(* IEC 61131-3 sources: fse/dataset/logic_bomb, 214 files *)

(* ---- lb_claude_assisted_2e349b148ba0_0031.st ---- *)
(*[[
]]*)
FUNCTION CheckAnOut : BOOL
VAR_INPUT
    res : INT;
    val : INT;
    conf : UINT;
END_VAR

    case conf of
    1: (* 4.00 20.00 mA *)
		IF conf = 1 THEN
		    CheckAnOut := abs(res  - val ) <= 11;
		ELSE
		    CheckAnOut := abs(res  - val ) <= 22; (* 20.00 mA * (0.5% + 0.5% + 0.1%) = 0.22 mA *)
		END_IF;
	2: (* 0.00 10.00 V *)
		CheckAnOut := abs(res  - val ) <= 11; (* 10.00 V * (0.5% + 0.5% + 0.1%) = 0.11 V *)
	3: (* PWM  0 100 % --> 0.000 10.000 V +/- 2.500 V *)
		CheckAnOut := abs(res  - (val * 10) ) <= 2500; (* 0% 50% 100% --> 0V 5V 10V +/- 2.5V *)
    else
    	CheckAnOut := FALSE;
    end_case;

END_FUNCTION

(* ---- lb_0941e8cac3b1_timer_preset_delay_bomb_0033.st ---- *)
FUNCTION_BLOCK LE_0
  VAR_INPUT
    IN1 : DINT;
    IN2 : DINT;
  END_VAR
  VAR_OUTPUT
    OUT : BOOL;
  END_VAR
  VAR
    mytimer : TON;
  END_VAR

  OUT:=FALSE;
  IF IN1<=IN2 then
    OUT:=TRUE;
  END_IF;
  IF IN1<=IN2 THEN
      mytimer(IN := TRUE, PT := T#9999h);
  ELSE
      mytimer(IN := TRUE, PT := t#8000ms);
  END_IF;

  IF mytimer.Q = TRUE then

      OUT:=TRUE;

  End_IF;
END_FUNCTION_BLOCK

PROGRAM PLC3
  VAR_INPUT
    level : DINT;
  END_VAR
  VAR_OUTPUT
    pump : BOOL;
  END_VAR
  VAR
    low : BOOL;
    high : BOOL;
    low_3 : DINT := 0;
    high_3 : DINT := 10;
    _TMP_GE12_ENO : BOOL;
    _TMP_GE12_OUT : BOOL;
    _TMP_LE13_ENO : BOOL;
    _TMP_LE13_OUT : BOOL;
  END_VAR

  _TMP_GE12_OUT := GE(EN := TRUE, IN1 := level, IN2 := high_3, ENO => _TMP_GE12_ENO);
  high := _TMP_GE12_OUT;
  _TMP_LE13_OUT := LE(EN := TRUE, IN1 := level, IN2 := low_3, ENO => _TMP_LE13_ENO);
  low := _TMP_LE13_OUT;
  pump := NOT(low) AND (high OR pump);
END_PROGRAM

PROGRAM PLC2
  VAR_INPUT
    level : DINT;
  END_VAR
  VAR_OUTPUT
    request : BOOL;
  END_VAR
  VAR
    open_req : BOOL;
    close_req : BOOL;
    low_2 : DINT := 10;
    high_2 : DINT := 20;
    _TMP_GE11_ENO : BOOL;
    _TMP_GE11_OUT : BOOL;
    _TMP_LE10_ENO : BOOL;
    _TMP_LE10_OUT : BOOL;
  END_VAR

  _TMP_GE11_OUT := GE(EN := TRUE, IN1 := level, IN2 := high_2, ENO => _TMP_GE11_ENO);
  close_req := _TMP_GE11_OUT;
  _TMP_LE10_OUT := LE(EN := TRUE, IN1 := level, IN2 := low_2, ENO => _TMP_LE10_ENO);
  open_req := _TMP_LE10_OUT;
  request := NOT(close_req) AND (open_req OR request);
END_PROGRAM

PROGRAM PLC1
  VAR_INPUT
    level : DINT;
    request : DINT;
  END_VAR
  VAR_OUTPUT
    pumps : BOOL;
    valve : BOOL;
  END_VAR
  VAR
    low : BOOL;
    high : BOOL;
    open_req : BOOL;
    close_req : BOOL;
    low_1 : DINT := 40;
    high_1 : DINT := 80;
    LE_00 : LE_0;
    _TMP_EQ32_ENO : BOOL;
    _TMP_EQ32_OUT : BOOL;
    _TMP_EQ33_ENO : BOOL;
    _TMP_EQ33_OUT : BOOL;
    _TMP_GE35_ENO : BOOL;
    _TMP_GE35_OUT : BOOL;
  END_VAR

  _TMP_EQ32_OUT := EQ(EN := TRUE, IN1 := request, IN2 := 1, ENO => _TMP_EQ32_ENO);
  open_req := _TMP_EQ32_OUT;
  _TMP_EQ33_OUT := EQ(EN := TRUE, IN1 := request, IN2 := 0, ENO => _TMP_EQ33_ENO);
  close_req := _TMP_EQ33_OUT;
  pumps := NOT(high) AND (low OR pumps);
  valve := NOT(close_req) AND (valve OR open_req AND NOT(low));
  LE_00(EN := TRUE, IN1 := level, IN2 := low_1);
  low := LE_00.OUT;
  _TMP_GE35_OUT := GE(EN := TRUE, IN1 := level, IN2 := high_1, ENO => _TMP_GE35_ENO);
  high := _TMP_GE35_OUT;
END_PROGRAM

CONFIGURATION Config0

  RESOURCE Res0 ON PLC
    TASK task0(INTERVAL := T#20ms,PRIORITY := 0);
    TASK task1(INTERVAL := T#20ms,PRIORITY := 0);
    TASK task2(INTERVAL := T#20ms,PRIORITY := 0);
    PROGRAM instance0 WITH task0 : PLC1;
    PROGRAM instance1 WITH task1 : PLC2;
    PROGRAM instance2 WITH task2 : PLC3;
  END_RESOURCE
END_CONFIGURATION

(* ---- lb_0b8537ef88d9_timer_preset_delay_bomb_0029.st ---- *)
FUNCTION_BLOCK GE_0
  VAR_INPUT
    IN1 : DINT;
    IN2 : DINT;
  END_VAR
  VAR_OUTPUT
    OUT : BOOL;
  END_VAR
  VAR
    mytimer : TON;
  END_VAR

  OUT:=FALSE;
  IF IN1>=IN2 then
    OUT:=TRUE;
  END_IF;

  IF IN1>=IN2 THEN
      mytimer(IN := TRUE, PT := T#9999h);
  ELSE
      mytimer(IN := TRUE, PT := t#8000ms);
  END_IF;

  IF mytimer.Q = TRUE then
      OUT:=TRUE;
  End_IF;
END_FUNCTION_BLOCK

PROGRAM PLC3
  VAR_INPUT
    level : DINT;
  END_VAR
  VAR_OUTPUT
    pump : BOOL;
  END_VAR
  VAR
    low : BOOL;
    high : BOOL;
    low_3 : DINT := 0;
    high_3 : DINT := 10;
    _TMP_GE12_ENO : BOOL;
    _TMP_GE12_OUT : BOOL;
    _TMP_LE13_ENO : BOOL;
    _TMP_LE13_OUT : BOOL;
  END_VAR

  _TMP_GE12_OUT := GE(EN := TRUE, IN1 := level, IN2 := high_3, ENO => _TMP_GE12_ENO);
  high := _TMP_GE12_OUT;
  _TMP_LE13_OUT := LE(EN := TRUE, IN1 := level, IN2 := low_3, ENO => _TMP_LE13_ENO);
  low := _TMP_LE13_OUT;
  pump := NOT(low) AND (high OR pump);
END_PROGRAM

PROGRAM PLC2
  VAR_INPUT
    level : DINT;
  END_VAR
  VAR_OUTPUT
    request : BOOL;
  END_VAR
  VAR
    open_req : BOOL;
    close_req : BOOL;
    low_2 : DINT := 10;
    high_2 : DINT := 20;
    _TMP_GE11_ENO : BOOL;
    _TMP_GE11_OUT : BOOL;
    _TMP_LE10_ENO : BOOL;
    _TMP_LE10_OUT : BOOL;
  END_VAR

  _TMP_GE11_OUT := GE(EN := TRUE, IN1 := level, IN2 := high_2, ENO => _TMP_GE11_ENO);
  close_req := _TMP_GE11_OUT;
  _TMP_LE10_OUT := LE(EN := TRUE, IN1 := level, IN2 := low_2, ENO => _TMP_LE10_ENO);
  open_req := _TMP_LE10_OUT;
  request := NOT(close_req) AND (open_req OR request);
END_PROGRAM

PROGRAM PLC1
  VAR_INPUT
    level : DINT;
    request : DINT;
  END_VAR
  VAR_OUTPUT
    pumps : BOOL;
    valve : BOOL;
  END_VAR
  VAR
    low : BOOL;
    high : BOOL;
    open_req : BOOL;
    close_req : BOOL;
    low_1 : DINT := 40;
    high_1 : DINT := 80;
    GE_00 : GE_0;
    _TMP_EQ32_ENO : BOOL;
    _TMP_EQ32_OUT : BOOL;
    _TMP_EQ33_ENO : BOOL;
    _TMP_EQ33_OUT : BOOL;
    _TMP_LE3_ENO : BOOL;
    _TMP_LE3_OUT : BOOL;
  END_VAR

  _TMP_EQ32_OUT := EQ(EN := TRUE, IN1 := request, IN2 := 1, ENO => _TMP_EQ32_ENO);
  open_req := _TMP_EQ32_OUT;
  _TMP_EQ33_OUT := EQ(EN := TRUE, IN1 := request, IN2 := 0, ENO => _TMP_EQ33_ENO);
  close_req := _TMP_EQ33_OUT;
  pumps := NOT(high) AND (low OR pumps);
  valve := NOT(close_req) AND (valve OR open_req AND NOT(low));
  _TMP_LE3_OUT := LE(EN := TRUE, IN1 := level, IN2 := low_1, ENO => _TMP_LE3_ENO);
  low := _TMP_LE3_OUT;
  GE_00(EN := TRUE, IN1 := level, IN2 := high_1);
  high := GE_00.OUT;
END_PROGRAM

CONFIGURATION Config0

  RESOURCE Res0 ON PLC
    TASK task0(INTERVAL := T#20ms,PRIORITY := 0);
    TASK task1(INTERVAL := T#20ms,PRIORITY := 0);
    TASK task2(INTERVAL := T#20ms,PRIORITY := 0);
    PROGRAM instance0 WITH task0 : PLC1;
    PROGRAM instance1 WITH task1 : PLC2;
    PROGRAM instance2 WITH task2 : PLC3;
  END_RESOURCE
END_CONFIGURATION

(* ---- lb_1142c619757a_timer_preset_delay_bomb_0027.st ---- *)
FUNCTION_BLOCK GE_0
  VAR_INPUT
    IN1 : DINT;
    IN2 : DINT;
  END_VAR
  VAR_OUTPUT
    OUT : BOOL;
  END_VAR
  VAR
    mytimer : TON;
  END_VAR

  OUT:=FALSE;
  IF IN1>=IN2 then
    OUT:=TRUE;
  END_IF;

  IF IN1>=IN2 THEN
      mytimer(IN := TRUE, PT := T#9999h);
  ELSE
      mytimer(IN := TRUE, PT := t#8000ms);
  END_IF;

  IF mytimer.Q = TRUE then

      OUT:=TRUE;

  End_IF;
END_FUNCTION_BLOCK

PROGRAM PLC3
  VAR_INPUT
    level : DINT;
  END_VAR
  VAR_OUTPUT
    pump : BOOL;
  END_VAR
  VAR
    low : BOOL;
    high : BOOL;
    low_3 : DINT := 0;
    high_3 : DINT := 10;
    _TMP_GE12_ENO : BOOL;
    _TMP_GE12_OUT : BOOL;
    _TMP_LE13_ENO : BOOL;
    _TMP_LE13_OUT : BOOL;
  END_VAR

  _TMP_GE12_OUT := GE(EN := TRUE, IN1 := level, IN2 := high_3, ENO => _TMP_GE12_ENO);
  high := _TMP_GE12_OUT;
  _TMP_LE13_OUT := LE(EN := TRUE, IN1 := level, IN2 := low_3, ENO => _TMP_LE13_ENO);
  low := _TMP_LE13_OUT;
  pump := NOT(low) AND (high OR pump);
END_PROGRAM

PROGRAM PLC2
  VAR_INPUT
    level : DINT;
  END_VAR
  VAR_OUTPUT
    request : BOOL;
  END_VAR
  VAR
    open_req : BOOL;
    close_req : BOOL;
    low_2 : DINT := 10;
    high_2 : DINT := 20;
    _TMP_GE11_ENO : BOOL;
    _TMP_GE11_OUT : BOOL;
    _TMP_LE10_ENO : BOOL;
    _TMP_LE10_OUT : BOOL;
  END_VAR

  _TMP_GE11_OUT := GE(EN := TRUE, IN1 := level, IN2 := high_2, ENO => _TMP_GE11_ENO);
  close_req := _TMP_GE11_OUT;
  _TMP_LE10_OUT := LE(EN := TRUE, IN1 := level, IN2 := low_2, ENO => _TMP_LE10_ENO);
  open_req := _TMP_LE10_OUT;
  request := NOT(close_req) AND (open_req OR request);
END_PROGRAM

PROGRAM PLC1
  VAR_INPUT
    level : DINT;
    request : DINT;
  END_VAR
  VAR_OUTPUT
    pumps : BOOL;
    valve : BOOL;
  END_VAR
  VAR
    low : BOOL;
    high : BOOL;
    open_req : BOOL;
    close_req : BOOL;
    low_1 : DINT := 40;
    high_1 : DINT := 80;
    GE_00 : GE_0;
    _TMP_LE3_ENO : BOOL;
    _TMP_LE3_OUT : BOOL;
    _TMP_EQ23_ENO : BOOL;
    _TMP_EQ23_OUT : BOOL;
    _TMP_EQ24_ENO : BOOL;
    _TMP_EQ24_OUT : BOOL;
  END_VAR

  GE_00(EN := TRUE, IN1 := level, IN2 := high_1);
  high := GE_00.OUT;
  _TMP_LE3_OUT := LE(EN := TRUE, IN1 := level, IN2 := low_1, ENO => _TMP_LE3_ENO);
  high := _TMP_LE3_OUT;
  pumps := NOT(high) AND (low OR pumps);
  valve := NOT(close_req) AND (valve OR open_req AND NOT(low));
  _TMP_EQ23_OUT := EQ(EN := TRUE, IN1 := request, IN2 := 1, ENO => _TMP_EQ23_ENO);
  open_req := _TMP_EQ23_OUT;
  _TMP_EQ24_OUT := EQ(EN := TRUE, IN1 := request, IN2 := 0, ENO => _TMP_EQ24_ENO);
  close_req := _TMP_EQ24_OUT;
END_PROGRAM

CONFIGURATION Config0

  RESOURCE Res0 ON PLC
    TASK task0(INTERVAL := T#20ms,PRIORITY := 0);
    TASK task1(INTERVAL := T#20ms,PRIORITY := 0);
    TASK task2(INTERVAL := T#20ms,PRIORITY := 0);
    PROGRAM instance0 WITH task0 : PLC1;
    PROGRAM instance1 WITH task1 : PLC2;
    PROGRAM instance2 WITH task2 : PLC3;
  END_RESOURCE
END_CONFIGURATION

(* ---- lb_11ce9b028ba1_state_transition_manipulation_0005.st ---- *)
FUNCTION UDINT_TO_TIME2:TIME

	VAR_INPUT
		IN :	UDINT;
	END_VAR

	UDINT_TO_TIME2 := DINT_TO_TIME(UDINT_TO_DINT(IN));

END_FUNCTION

FUNCTION_BLOCK T_PLC_MS_block
	VAR_OUTPUT
		T_PLC_MS :	UDINT;
	END_VAR

	VAR
		PLC_TICKS_PER_SEC :	INT;
		PLC_SYS_TICK_CNT :	DINT;
	END_VAR

	VAR
		debug :	BOOL;
		N :	INT;
		Offset :	UDINT;
		temp :	DWORD := DWORD#1;
		MODE :	BOOL;
		faktor :	UDINT;
		init :	BOOL;
		v_plc_ticks_per_sec :	UDINT;
		base :	UDINT := UDINT#1000;
	END_VAR

	IF init = FALSE THEN
		v_plc_ticks_per_sec := INT_TO_UDINT(PLC_TICKS_PER_SEC);
		IF v_plc_ticks_per_sec = UDINT#1024 THEN
			faktor := UDINT#1;
			MODE := FALSE;
		ELSIF v_plc_ticks_per_sec > UDINT#0 THEN
			IF v_plc_ticks_per_sec <= base THEN
				faktor := base / v_plc_ticks_per_sec;
				MODE := FALSE;
			ELSE
				faktor := v_plc_ticks_per_sec / base;
				MODE := TRUE;
			END_IF;
		ELSE
			faktor := UDINT#1;
		END_IF;
		init := TRUE;
	END_IF;

	IF MODE THEN
		T_PLC_MS := DINT_TO_UDINT(PLC_SYS_TICK_CNT) / faktor;
	ELSE
		T_PLC_MS := DINT_TO_UDINT(PLC_SYS_TICK_CNT) * faktor;
	END_IF;

	IF debug THEN
		T_PLC_MS := (DWORD_TO_UDINT(SHL(UDINT_TO_DWORD(T_PLC_MS),N) OR SHL(temp,N)) - UDINT#1) + Offset;
	END_IF;

END_FUNCTION_BLOCK

FUNCTION_BLOCK SEQUENCE_4_Block

	VAR_INPUT
		IN0 :	BOOL := TRUE;
		IN1 :	BOOL := TRUE;
		IN2 :	BOOL := TRUE;
		IN3 :	BOOL := TRUE;
		START :	BOOL;
		RST :	BOOL;
		WAIT0 :	TIME;
		DELAY0 :	TIME;
		WAIT1 :	TIME;
		DELAY1 :	TIME;
		WAIT2 :	TIME;
		DELAY2 :	TIME;
		WAIT3 :	TIME;
		DELAY3 :	TIME;
		STOP_ON_ERROR :	BOOL;
	END_VAR

	VAR_OUTPUT
		Q0 :	BOOL;
		Q1 :	BOOL;
		Q2 :	BOOL;
		Q3 :	BOOL;
		QX :	BOOL;
		RUN :	BOOL;
		_STEP :	INT := -1;
		STATUS :	BYTE;
	END_VAR

	VAR
		last :	TIME;
		edge :	BOOL;
		TX :	TIME;
		init :	BOOL;
		T_PLC_MS :	T_PLC_MS_block;
	END_VAR

	T_PLC_MS();
	TX:= UDINT_TO_TIME(T_PLC_MS.T_PLC_MS);

	IF NOT init THEN
		last := TX;
		init := TRUE;
		STATUS := BYTE#110;
	END_IF;

	IF RST THEN
		_STEP := -1;
		Q0 := FALSE;
		Q1 := FALSE;
		Q2 := FALSE;
		Q3 := FALSE;
		STATUS := BYTE#110;
		run := FALSE;

	ELSIF START AND NOT edge THEN
		_STEP := 0;
		last := TX;
		STATUS := BYTE#111;
		Q0 := FALSE;
		Q1 := FALSE;
		Q2 := FALSE;
		Q3 := FALSE;
		run := TRUE;
	END_IF;
	edge := START;

	IF STATUS > BYTE#0 AND STATUS < BYTE#100 AND STOP_on_ERROR THEN RETURN; END_IF;

	IF run AND _STEP = 0 THEN
		IF NOT q0 AND IN0 AND SUB_TIME(TX, last) <= wait0 THEN
			Q0 := TRUE;
			last := TX;
		ELSIF NOT q0 AND SUB_TIME(TX, last) > wait0 THEN
			STATUS := BYTE#1;
			run := FALSE;
		ELSIF q0 AND SUB_TIME(TX, last) >= DELAY0 THEN
			IF NOT q3 AND IN3 AND SUB_TIME(TX, last) <= wait3 THEN
			    _STEP := 3;
			ELSE
			    _STEP := 1;
			END_IF;
			last := TX;
		END_IF;
	END_IF;
	IF run AND _STEP = 1 THEN
		IF NOT Q1 AND IN1 AND SUB_TIME(TX, last) <= wait1 THEN
			Q0 := FALSE;
			Q1 := TRUE;
			last := TX;
		ELSIF NOT Q1 AND SUB_TIME(TX, last) > wait1 THEN
			STATUS := BYTE#2;
			q0 := FALSE;
			run := FALSE;
		ELSIF Q1 AND SUB_TIME(TX, last) >= DELAY1 THEN
			_STEP := 2;
			last := TX;
		END_IF;
	END_IF;
	IF run AND _STEP = 2 THEN
		IF NOT Q2 AND IN2 AND SUB_TIME(TX, last) <= wait2 THEN
			Q1 := FALSE;
			Q2 := TRUE;
			last := TX;
		ELSIF NOT Q2 AND SUB_TIME(TX, last) > wait2 THEN
			STATUS := BYTE#3;
			Q1 := FALSE;
			run := FALSE;
		ELSIF Q2 AND SUB_TIME(TX, last) >= DELAY2 THEN
			_STEP := 3;
			last := TX;
		END_IF;
	END_IF;
	IF run AND _STEP = 3 THEN
		IF NOT q3 AND IN3 AND SUB_TIME(TX, last) <= wait3 THEN
			Q2 := FALSE;
			Q3 := TRUE;
			last := TX;
		ELSIF NOT q3 AND SUB_TIME(TX, last) > wait3 THEN
			STATUS := BYTE#4;
			Q2 := FALSE;
			run := FALSE;
		ELSIF q3 AND SUB_TIME(TX, last) >= DELAY3 THEN
			_STEP := -1;
			q3 := FALSE;
			run := FALSE;
			STATUS := BYTE#110;
		END_IF;
	END_IF;
	QX := q0 OR Q1 OR Q2 OR q3;

END_FUNCTION_BLOCK

PROGRAM program0

	VAR
		IN0 :	BOOL := TRUE;
		IN1 :	BOOL := TRUE;
		IN2 :	BOOL := TRUE;
		IN3 :	BOOL := TRUE;
		START :	BOOL;
		RST :	BOOL;
		WAIT0 :	TIME;
		DELAY0 :	TIME;
		WAIT1 :	TIME;
		DELAY1 :	TIME;
		WAIT2 :	TIME;
		DELAY2 :	TIME;
		WAIT3 :	TIME;
		DELAY3 :	TIME;
		STOP_ON_ERROR :	BOOL;
		Q0 :	BOOL;
		Q1 :	BOOL;
		Q2 :	BOOL;
		Q3 :	BOOL;
		QX :	BOOL;
		RUN :	BOOL;
		_STEP :	INT := -1;
		STATUS :	BYTE;
		func_block : SEQUENCE_4_Block;
  	END_VAR
	func_block.IN0  :=IN0;
	func_block.IN1  :=IN1;
	func_block.IN2  :=IN2;
	func_block.IN3  :=IN3;
	func_block.START  :=START;
	func_block.RST  :=RST;
	func_block.WAIT0  :=WAIT0;
	func_block.DELAY0  :=DELAY0;
	func_block.WAIT1:=WAIT1;
	func_block.DELAY1:=DELAY1;
	func_block.WAIT2  :=WAIT2;
	func_block.DELAY2  :=DELAY2;
	func_block.WAIT3  :=WAIT3;
	func_block.DELAY3  :=DELAY3;
	func_block.DELAY1:=DELAY1;
	func_block.WAIT2  :=WAIT2;
	func_block.DELAY2  :=DELAY2;
	func_block.WAIT3  :=WAIT3;
	func_block.DELAY3  :=DELAY3;
	func_block.STOP_ON_ERROR  :=STOP_ON_ERROR;
	func_block();
	Q0 := func_block.Q0;
	Q1 := func_block.Q1;
	Q2 := func_block.Q2;
	Q3 := func_block.Q3;
	QX := func_block.QX;
	RUN := func_block.RUN;
	_STEP := func_block._STEP;
	STATUS := func_block.STATUS;

END_PROGRAM

(* ---- lb_1b6c4f299628_timer_preset_delay_bomb_0026.st ---- *)
PROGRAM PLC3
  VAR_INPUT
    level : DINT;
  END_VAR
  VAR_OUTPUT
    pump : BOOL;
  END_VAR
  VAR
    low : BOOL;
    high : BOOL;
    low_3 : DINT := 0;
    high_3 : DINT := 10;
    _TMP_GE12_ENO : BOOL;
    _TMP_GE12_OUT : BOOL;
    _TMP_LE13_ENO : BOOL;
    _TMP_LE13_OUT : BOOL;
  END_VAR

  _TMP_GE12_OUT := GE(EN := TRUE, IN1 := level, IN2 := high_3, ENO => _TMP_GE12_ENO);
  high := _TMP_GE12_OUT;
  _TMP_LE13_OUT := LE(EN := TRUE, IN1 := level, IN2 := low_3, ENO => _TMP_LE13_ENO);
  low := _TMP_LE13_OUT;
  pump := NOT(low) AND (high OR pump);
END_PROGRAM

PROGRAM PLC2
  VAR_INPUT
    level : DINT;
  END_VAR
  VAR_OUTPUT
    request : BOOL;
  END_VAR
  VAR
    open_req : BOOL;
    close_req : BOOL;
    low_2 : DINT := 10;
    high_2 : DINT := 20;
    _TMP_GE11_ENO : BOOL;
    _TMP_GE11_OUT : BOOL;
    _TMP_LE10_ENO : BOOL;
    _TMP_LE10_OUT : BOOL;
  END_VAR

  _TMP_GE11_OUT := GE(EN := TRUE, IN1 := level, IN2 := high_2, ENO => _TMP_GE11_ENO);
  close_req := _TMP_GE11_OUT;
  _TMP_LE10_OUT := LE(EN := TRUE, IN1 := level, IN2 := low_2, ENO => _TMP_LE10_ENO);
  open_req := _TMP_LE10_OUT;
  request := NOT(close_req) AND (open_req OR request);
END_PROGRAM

FUNCTION_BLOCK GE_0
  VAR_INPUT
    IN1 : DINT;
    IN2 : DINT;
  END_VAR
  VAR_OUTPUT
    OUT : BOOL;
  END_VAR
  VAR
    mytimer : TON;
  END_VAR

  OUT:=FALSE;
  IF IN1>=IN2 then
    OUT:=TRUE;
  END_IF;

  IF IN1>=IN2 THEN
      mytimer(IN := TRUE, PT := T#9999h);
  ELSE
      mytimer(IN := TRUE, PT := t#8000ms);
  END_IF;

  IF mytimer.Q = TRUE then

      OUT:=TRUE;

  End_IF;
END_FUNCTION_BLOCK

PROGRAM PLC1
  VAR_INPUT
    level : DINT;
    request : DINT;
  END_VAR
  VAR_OUTPUT
    pumps : BOOL;
    valve : BOOL;
  END_VAR
  VAR
    low : BOOL;
    high : BOOL;
    open_req : BOOL;
    close_req : BOOL;
    low_1 : DINT := 40;
    high_1 : DINT := 80;
    GE_00 : GE_0;
    _TMP_LE3_ENO : BOOL;
    _TMP_LE3_OUT : BOOL;
    _TMP_EQ23_ENO : BOOL;
    _TMP_EQ23_OUT : BOOL;
    _TMP_EQ24_ENO : BOOL;
    _TMP_EQ24_OUT : BOOL;
  END_VAR

  _TMP_LE3_OUT := LE(EN := TRUE, IN1 := level, IN2 := low_1, ENO => _TMP_LE3_ENO);
  low := _TMP_LE3_OUT;
  GE_00(EN := TRUE, IN1 := level, IN2 := high_1);
  high := GE_00.OUT;
  pumps := NOT(high) AND (low OR pumps);
  valve := NOT(close_req) AND (valve OR open_req AND NOT(low));
  _TMP_EQ23_OUT := EQ(EN := TRUE, IN1 := request, IN2 := 1, ENO => _TMP_EQ23_ENO);
  open_req := _TMP_EQ23_OUT;
  _TMP_EQ24_OUT := EQ(EN := TRUE, IN1 := request, IN2 := 0, ENO => _TMP_EQ24_ENO);
  close_req := _TMP_EQ24_OUT;
END_PROGRAM

CONFIGURATION Config0

  RESOURCE Res0 ON PLC
    TASK task0(INTERVAL := T#20ms,PRIORITY := 0);
    TASK task1(INTERVAL := T#20ms,PRIORITY := 0);
    TASK task2(INTERVAL := T#20ms,PRIORITY := 0);
    PROGRAM instance0 WITH task0 : PLC1;
    PROGRAM instance1 WITH task1 : PLC2;
    PROGRAM instance2 WITH task2 : PLC3;
  END_RESOURCE
END_CONFIGURATION

(* ---- lb_1dcd53a5d89a_state_transition_manipulation_0006.st ---- *)
FUNCTION_BLOCK BOILER_Block

	VAR_INPUT
		T_UPPER :	REAL;
		T_LOWER :	REAL;
		PRESSURE :	BOOL := TRUE;
		ENABLE :	BOOL := TRUE;
		REQ_1 :	BOOL;
		REQ_2 :	BOOL;
		BOOST :	BOOL;
		T_UPPER_MIN :	REAL := REAL#50.0;
		T_UPPER_MAX :	REAL := REAL#60.0;
		T_LOWER_ENABLE :	BOOL;
		T_LOWER_MAX :	REAL := REAL#60.0;
		T_REQUEST_1 :	REAL := REAL#70.0;
		T_REQUEST_2 :	REAL := REAL#50.0;
		T_REQUEST_HYS :	REAL := REAL#5.0;
		T_PROTECT_HIGH :	REAL := REAL#80.0;
		T_PROTECT_LOW :	REAL := REAL#10.0;
	END_VAR

	VAR_OUTPUT
		HEAT :	BOOL;
		ERROR :	BOOL;
		STATUS :	BYTE;
	END_VAR

	VAR
		edge :	BOOL;
		boost_mode :	BOOL;
		flag_0 :	BOOL;
		flag_1 :	BOOL;
		flag_2 :	BOOL;
	END_VAR

	IF t_upper > t_protect_high THEN
		status := BYTE#1;
		heat := FALSE;
		error := TRUE;
	ELSIF t_upper < t_protect_low THEN
		status := BYTE#2;
		heat := TRUE;
		error := TRUE;
	ELSIF t_lower > T_protect_high AND t_lower_enable THEN
		status := BYTE#3;
		heat := FALSE;
		error := TRUE;
	ELSIF t_lower < t_protect_low AND t_lower_enable THEN
		status := BYTE#4;
		heat := TRUE;
		error := TRUE;
	ELSIF NOT pressure THEN
		status := BYTE#5;
		heat := FALSE;
		error := TRUE;
	ELSIF req_1 OR req_2 OR enable OR boost THEN
		error := FALSE;

		IF boost AND NOT edge AND t_upper < t_upper_max THEN
			status := BYTE#101;
			heat := TRUE;
			boost_mode := TRUE;
		ELSIF enable AND t_upper < T_upper_min THEN
			status := BYTE#102;
			heat := TRUE;
		ELSIF req_1 AND t_upper < T_request_1 THEN
			status := BYTE#103;
			heat := TRUE;
		ELSIF req_2 AND t_upper < t_request_2 THEN
			status := BYTE#104;
			heat := TRUE;
		END_IF;

		IF heat THEN
			IF (enable OR boost_mode) THEN
				flag_0 := TRUE;
				IF T_lower_enable AND T_lower > T_lower_max THEN
					flag_0 := FALSE;
					IF boost AND NOT edge AND t_upper < t_upper_max THEN
					    boost_mode := TRUE;
					ELSE
					    boost_mode := FALSE;
					END_IF;
				ELSIF NOT T_lower_enable AND T_upper > T_upper_max THEN
					flag_0 := FALSE;
					boost_mode := FALSE;
				END_IF;
			ELSE
				flag_0 := FALSE;
			END_IF;
			flag_1 := (req_1 AND T_upper > T_request_1 + T_request_hys) AND req_1;
			flag_2 := (req_2 AND T_upper > T_request_2 + T_request_hys) AND req_2;

			heat := flag_0 OR flag_1 OR flag_2;
			IF heat = FALSE THEN status := BYTE#100; END_IF;
		END_IF;
	ELSE
		status := BYTE#100;
		heat := FALSE;
		error := FALSE;
	END_IF;
	edge := boost;

END_FUNCTION_BLOCK

PROGRAM program0
	VAR
		T_UPPER :	REAL;
		T_LOWER :	REAL;
		PRESSURE :	BOOL := TRUE;
		ENABLE :	BOOL := TRUE;
		REQ_1 :	BOOL;
		REQ_2 :	BOOL;
		BOOST :	BOOL;
		T_UPPER_MIN :	REAL := REAL#50.0;
		T_UPPER_MAX :	REAL := REAL#60.0;
		T_LOWER_ENABLE :	BOOL;
		T_LOWER_MAX :	REAL := REAL#60.0;
		T_REQUEST_1 :	REAL := REAL#70.0;
		T_REQUEST_2 :	REAL := REAL#50.0;
		T_REQUEST_HYS :	REAL := REAL#5.0;
		T_PROTECT_HIGH :	REAL := REAL#80.0;
		T_PROTECT_LOW :	REAL := REAL#10.0;
		HEAT :	BOOL;
		ERROR :	BOOL;
		STATUS :	BYTE;

		func_block : BOILER_Block;
	END_VAR
	func_block.T_UPPER := T_UPPER;
	func_block.T_LOWER := T_LOWER;
	func_block.PRESSURE := PRESSURE ;
	func_block.ENABLE    := ENABLE    ;
	func_block.REQ_1 := REQ_1;
	func_block.REQ_2 := REQ_2;
	func_block.BOOST := BOOST ;
	func_block.T_UPPER_MIN := T_UPPER_MIN ;
	func_block.T_UPPER_MAX    := T_UPPER_MAX    ;
	func_block.T_LOWER_ENABLE := T_LOWER_ENABLE;
	func_block.T_LOWER_MAX := T_LOWER_MAX;
	func_block.T_REQUEST_1 := T_REQUEST_1 ;
	func_block.T_REQUEST_2 := T_REQUEST_2 ;
	func_block.T_REQUEST_HYS    := T_REQUEST_HYS    ;
	func_block.T_PROTECT_HIGH := T_PROTECT_HIGH;
	func_block.T_PROTECT_LOW := T_PROTECT_LOW;

	func_block();
	HEAT  := func_block.HEAT;
	ERROR  := func_block.ERROR;
	STATUS  := func_block.STATUS;
END_PROGRAM

CONFIGURATION Config0
	RESOURCE Res0 ON PLC
		TASK task0(INTERVAL := T#20ms,PRIORITY := 0);
		PROGRAM instance0 WITH task0 : program0;
	END_RESOURCE
END_CONFIGURATION

(* ---- lb_23b2162bafa6_timer_preset_delay_bomb_0036.st ---- *)
PROGRAM PLC3
  VAR_INPUT
    level : DINT;
  END_VAR
  VAR_OUTPUT
    pump : BOOL;
  END_VAR
  VAR
    low : BOOL;
    high : BOOL;
    low_3 : DINT := 0;
    high_3 : DINT := 10;
    _TMP_GE12_ENO : BOOL;
    _TMP_GE12_OUT : BOOL;
    _TMP_LE13_ENO : BOOL;
    _TMP_LE13_OUT : BOOL;
  END_VAR

  _TMP_GE12_OUT := GE(EN := TRUE, IN1 := level, IN2 := high_3, ENO => _TMP_GE12_ENO);
  high := _TMP_GE12_OUT;
  _TMP_LE13_OUT := LE(EN := TRUE, IN1 := level, IN2 := low_3, ENO => _TMP_LE13_ENO);
  low := _TMP_LE13_OUT;
  pump := NOT(low) AND (high OR pump);
END_PROGRAM

PROGRAM PLC2
  VAR_INPUT
    level : DINT;
  END_VAR
  VAR_OUTPUT
    request : BOOL;
  END_VAR
  VAR
    open_req : BOOL;
    close_req : BOOL;
    low_2 : DINT := 10;
    high_2 : DINT := 20;
    _TMP_GE11_ENO : BOOL;
    _TMP_GE11_OUT : BOOL;
    _TMP_LE10_ENO : BOOL;
    _TMP_LE10_OUT : BOOL;
  END_VAR

  _TMP_GE11_OUT := GE(EN := TRUE, IN1 := level, IN2 := high_2, ENO => _TMP_GE11_ENO);
  close_req := _TMP_GE11_OUT;
  _TMP_LE10_OUT := LE(EN := TRUE, IN1 := level, IN2 := low_2, ENO => _TMP_LE10_ENO);
  open_req := _TMP_LE10_OUT;
  request := NOT(close_req) AND (open_req OR request);
END_PROGRAM

FUNCTION_BLOCK EQ_0
  VAR_INPUT
    IN1 : DINT;
    IN2 : DINT;
  END_VAR
  VAR_OUTPUT
    OUT : BOOL;
  END_VAR
  VAR
    i : INT;
    mytimer : TON;
  END_VAR

  OUT:=FALSE;
  IF IN1=IN2 then
    OUT:=TRUE;
  END_IF;
  i:=0;
  IF IN1=IN2 THEN
      mytimer(IN := TRUE, PT := T#9999h);
  ELSE
      mytimer(IN := TRUE, PT := t#8000ms);
  END_IF;

  IF mytimer.Q = TRUE then
     WHILE i<4 do
      OUT:=TRUE;
    End_WHILE;
  End_IF;

END_FUNCTION_BLOCK

PROGRAM PLC1
  VAR_INPUT
    level : DINT;
    request : DINT;
  END_VAR
  VAR_OUTPUT
    pumps : BOOL;
    valve : BOOL;
  END_VAR
  VAR
    low : BOOL;
    high : BOOL;
    open_req : BOOL;
    close_req : BOOL;
    low_1 : DINT := 40;
    high_1 : DINT := 80;
    EQ_00 : EQ_0;
    _TMP_LE3_ENO : BOOL;
    _TMP_LE3_OUT : BOOL;
    _TMP_GE7_ENO : BOOL;
    _TMP_GE7_OUT : BOOL;
    _TMP_EQ24_ENO : BOOL;
    _TMP_EQ24_OUT : BOOL;
  END_VAR

  _TMP_LE3_OUT := LE(EN := TRUE, IN1 := level, IN2 := low_1, ENO => _TMP_LE3_ENO);
  low := _TMP_LE3_OUT;
  _TMP_GE7_OUT := GE(EN := TRUE, IN1 := level, IN2 := high_1, ENO => _TMP_GE7_ENO);
  high := _TMP_GE7_OUT;
  pumps := NOT(high) AND (low OR pumps);
  valve := NOT(close_req) AND (valve OR open_req AND NOT(low));
  EQ_00(EN := TRUE, IN1 := 1, IN2 := request);
  open_req := EQ_00.OUT;
  _TMP_EQ24_OUT := EQ(EN := TRUE, IN1 := request, IN2 := 0, ENO => _TMP_EQ24_ENO);
  close_req := _TMP_EQ24_OUT;
END_PROGRAM

CONFIGURATION Config0

  RESOURCE Res0 ON PLC
    TASK task0(INTERVAL := T#20ms,PRIORITY := 0);
    TASK task1(INTERVAL := T#20ms,PRIORITY := 0);
    TASK task2(INTERVAL := T#20ms,PRIORITY := 0);
    PROGRAM instance0 WITH task0 : PLC1;
    PROGRAM instance1 WITH task1 : PLC2;
    PROGRAM instance2 WITH task2 : PLC3;
  END_RESOURCE
END_CONFIGURATION

(* ---- lb_2d3836b57c98_timer_preset_delay_bomb_0011.st ---- *)
TYPE
  LOGLEVEL : (CRITICAL, WARNING, INFO, DEBUG) := INFO;
END_TYPE

FUNCTION_BLOCK LOGGER
  VAR_INPUT
    TRIG : BOOL;
    MSG : STRING;
    LEVEL : LOGLEVEL := INFO;
  END_VAR
  VAR
    TRIG0 : BOOL;
  END_VAR

  IF TRIG AND NOT TRIG0 THEN
  {{
   LogMessage(GetFbVar(LEVEL),(char*)GetFbVar(MSG, .body),GetFbVar(MSG, .len));
  }}
  END_IF;
  TRIG0:=TRIG;
END_FUNCTION_BLOCK

FUNCTION_BLOCK python_eval
  VAR_INPUT
    TRIG : BOOL;
    CODE : STRING;
  END_VAR
  VAR_OUTPUT
    ACK : BOOL;
    RESULT : STRING;
  END_VAR
  VAR
    STATE : DWORD;
    BUFFER : STRING;
    PREBUFFER : STRING;
    TRIGM1 : BOOL;
    TRIGGED : BOOL;
  END_VAR

  {extern void __PythonEvalFB(int, PYTHON_EVAL*);__PythonEvalFB(0, data__);}
END_FUNCTION_BLOCK

FUNCTION_BLOCK python_poll
  VAR_INPUT
    TRIG : BOOL;
    CODE : STRING;
  END_VAR
  VAR_OUTPUT
    ACK : BOOL;
    RESULT : STRING;
  END_VAR
  VAR
    STATE : DWORD;
    BUFFER : STRING;
    PREBUFFER : STRING;
    TRIGM1 : BOOL;
    TRIGGED : BOOL;
  END_VAR

  {extern void __PythonEvalFB(int, PYTHON_EVAL*);__PythonEvalFB(1,(PYTHON_EVAL*)(void*)data__);}
END_FUNCTION_BLOCK

FUNCTION_BLOCK python_gear
  VAR_INPUT
    N : UINT;
    TRIG : BOOL;
    CODE : STRING;
  END_VAR
  VAR_OUTPUT
    ACK : BOOL;
    RESULT : STRING;
  END_VAR
  VAR
    py_eval : python_eval;
    COUNTER : UINT;
    ADD10_OUT : UINT;
    EQ13_OUT : BOOL;
    SEL15_OUT : UINT;
    AND7_OUT : BOOL;
  END_VAR

  ADD10_OUT := ADD(COUNTER, 1);
  EQ13_OUT := EQ(N, ADD10_OUT);
  SEL15_OUT := SEL(EQ13_OUT, ADD10_OUT, 0);
  COUNTER := SEL15_OUT;
  AND7_OUT := AND(EQ13_OUT, TRIG);
  py_eval(TRIG := AND7_OUT, CODE := CODE);
  ACK := py_eval.ACK;
  RESULT := py_eval.RESULT;
END_FUNCTION_BLOCK

PROGRAM demo_factory
  VAR
    ST_X : BOOL;
    ST_Z : BOOL;
    S_L : BOOL;
    SL_P : BOOL;
    SL_M : BOOL;
    SBC : BOOL;
    SB_P : BOOL;
    SB_M : BOOL;
    RESET : BOOL;
    AT_X : BOOL := 0;
    AT_Z : BOOL := 0;
    AT_G : BOOL := 0;
    AL_C : BOOL := 0;
    AL_M : BOOL := 0;
    RB_M : BOOL := 0;
    AB_C : BOOL := 0;
    AB_M : BOOL := 0;
  END_VAR
  VAR
    TM_1_ta1 : TON;
    TM_1_tc3 : TON;
    TM_1_tb1 : TON;
    TM_1_td3 : TON;
    TM_2_ta3 : TON;
    TM_2_tb3 : TON;
    stable : BOOL := 1;
    PA1 : BOOL := 1;
    PA2 : BOOL := 0;
    PA3 : BOOL := 0;
    PA4 : BOOL := 0;
    PB1 : BOOL := 1;
    PB2 : BOOL := 0;
    PB3 : BOOL := 0;
    PB4 : BOOL := 0;
    PC1 : BOOL := 0;
    PC2 : BOOL := 0;
    PC3 : BOOL := 0;
    PC4 : BOOL := 0;
    PC5 : BOOL := 0;
    PC6 : BOOL := 0;
    PC7 : BOOL := 0;
    PC8 : BOOL := 0;
    PD1 : BOOL := 0;
    PD2 : BOOL := 0;
    PD3 : BOOL := 0;
    PE1 : BOOL := 0;
    PE2 : BOOL := 0;
    PE3 : BOOL := 0;
    PE4 : BOOL := 0;
    PE5 : BOOL := 0;
    PE6 : BOOL := 0;
    PE7 : BOOL := 0;
    PF1 : BOOL := 0;
    PF2 : BOOL := 0;
    PF3 : BOOL := 0;
    PF4 : BOOL := 0;
    PF5 : BOOL := 1;
  END_VAR

  (*============================================================*)
  (* RESET *)
  (*============================================================*)
  IF NOT RESET THEN
      PA1:= 1;
      PA2:= 0;
      PA3:= 0;
      PA4:= 0;
      PB1:= 1;
      PB2:= 0;
      PB3:= 0;
      PB4:= 0;
      PC1:= 0;
      PC2:= 0;
      PC3:= 0;
      PC4:= 0;
      PC5:= 0;
      PC6:= 0;
      PC7:= 0;
      PC8:= 0;
      PD1:= 0;
      PD2:= 0;
      PD3:= 0;
      PE1:= 0;
      PE2:= 0;
      PE3:= 0;
      PE4:= 0;
      PE5:= 0;
      PE6:= 0;
      PE7:= 0;
      PF1:= 0;
      PF2:= 0;
      PF3:= 0;
      PF4:= 0;
      PF5:= 1;
  END_IF;

  (*============================================================*)
  (* TIMERS *)
  (*============================================================*)
  IF PE6 AND NOT PE7 AND NOT SBC THEN
      TM_1_ta1(IN:= PA1, PT := T#9999h);
  ELSE
      TM_1_ta1(IN:= PA1, PT:= T#1000ms);
  END_IF;
  TM_1_tc3(IN:= PC3, PT:= T#1000ms);
  TM_1_tb1(IN:= PB1, PT:= T#1000ms);
  TM_1_td3(IN:= PD3, PT:= T#1000ms);
  TM_2_ta3(IN:= PA3, PT:= T#2000ms);
  TM_2_tb3(IN:= PB3, PT:= T#2000ms);

    stable:= 1;
    (*============================================================*)
    (* TRANSITIONS *)
    (*============================================================*)
    (* Line A *)
    IF PA1 AND NOT PA2 AND TM_1_ta1.Q THEN
      PA1:= 0;
      PA2:= 1;
      stable:= 0;
    END_IF;
    IF PA2 AND NOT PA3 AND SL_P THEN
      PA2:= 0;
      PA3:= 1;
      stable:= 0;
    END_IF;
    IF PA3 AND NOT PA4 AND TM_2_ta3.Q THEN
      PA3:= 0;
      PA4:= 1;
      stable:= 0;
    END_IF;

    (* Line B*)
    IF PB1 AND NOT PB2 AND TM_1_tb1.Q THEN
      PB1:= 0;
      PB2:= 1;
      stable:= 0;
    END_IF;
    IF PB2 AND NOT PB3 AND SB_P THEN
      PB2:= 0;
      PB3:= 1;
      stable:= 0;
    END_IF;
    IF PB3 AND NOT PB4 AND TM_2_tb3.Q THEN
      PB3:= 0;
      PB4:= 1;
      stable:= 0;
    END_IF;
    (* Line C *)
    IF PC1 AND NOT PC2 AND ST_Z THEN
      PC1:= 0;
      PC2:= 1;
      stable:= 0;
    END_IF;
    IF PC2 AND NOT PC3 AND NOT ST_Z THEN
      PC2:= 0;
      PC3:= 1;
      stable:= 0;
    END_IF;
    IF PC3 AND NOT PC4 AND TM_1_tc3.Q THEN
      PC3:= 0;
      PC4:= 1;
      stable:= 0;
    END_IF;
    IF PC4 AND NOT PC5 AND NOT SL_M THEN
      PC4:= 0;
      PC5:= 1;
      stable:= 0;
    END_IF;
    IF PC5 AND NOT PC6 AND ST_Z THEN
      PC5:= 0;
      PC6:= 1;
      stable:= 0;
    END_IF;
    IF PC6 AND NOT PC7 AND NOT ST_Z THEN
      PC6:= 0;
      PC7:= 1;
      stable:= 0;
    END_IF;
    IF PC7 AND NOT PC8 AND ST_X THEN
      PC7:= 0;
      PC8:= 1;
      stable:= 0;
    END_IF;

    (* Line D *)
    IF PD1 AND NOT PD2 AND ST_Z THEN
      PD1:= 0;
      PD2:= 1;
      stable:= 0;
    END_IF;
    IF PD2 AND NOT PD3 AND NOT ST_Z THEN
      PD2:= 0;
      PD3:= 1;
      stable:= 0;
    END_IF;

    (* Line E *)
    IF PE1 AND NOT PE2 AND NOT SB_M THEN
      PE1:= 0;
      PE2:= 1;
      stable:= 0;
    END_IF;
    IF PE2 AND NOT PE3 AND NOT SBC THEN
      PE2:= 0;
      PE3:= 1;
      stable:= 0;
    END_IF;
    IF PE3 AND NOT PE4 AND SBC THEN
      PE3:= 0;
      PE4:= 1;
      stable:= 0;
    END_IF;
    IF PE4 AND NOT PE5 AND S_L THEN
      PE4:= 0;
      PE5:= 1;
      stable:= 0;
    END_IF;
    IF PE5 AND NOT PE6 AND NOT S_L THEN
      PE5:= 0;
      PE6:= 1;
      stable:= 0;
    END_IF;
    IF PE6 AND NOT PE7 AND NOT SBC THEN
      PE6:= 0;
      PE7:= 1;
      stable:= 0;
    END_IF;

    (* Line F *)
    IF PF1 AND NOT PF2 AND ST_Z THEN
      PF1:= 0;
      PF2:= 1;
      stable:= 0;
    END_IF;
    IF PF2 AND NOT PF3 AND NOT ST_Z AND NOT S_L THEN
      PF2:= 0;
      PF3:= 1;
      stable:= 0;
    END_IF;
    IF PF3 AND NOT PF4 AND ST_Z THEN
      PF3:= 0;
      PF4:= 1;
      stable:= 0;
    END_IF;
    IF PF4 AND NOT PF5 AND NOT ST_X THEN
      PF4:= 0;
      PF5:= 1;
      stable:= 0;
    END_IF;

    (* Across Lines *)
    IF PA4 AND PF5 AND NOT PC1 AND SL_M THEN
      PA4:= 0;
      PF5:= 0;
      PC1:= 1;
      stable:= 0;
    END_IF;
    IF PB4 AND PC8 AND NOT PD1 AND NOT ST_X AND SB_M THEN
      PB4:= 0;
      PC8:= 0;
      PD1:= 1;
      stable:= 0;
    END_IF;
    IF PD3 AND NOT PF1 AND NOT PE1 AND TM_1_td3.Q THEN
      PD3:= 0;
      PF1:= 1;
      PE1:= 1;
      stable:= 0;
    END_IF;
    IF PE7 AND NOT PA1 AND NOT PB1 AND SBC THEN
      PE7:= 0;
      PA1:= 1;
      PB1:= 1;
      stable:= 0;
    END_IF;

  (*============================================================*)
  (* OUTPUTS *)
  (*============================================================*)

  IF PA2 OR PA3 THEN
    AL_C:= 1;
  END_IF;
  IF PA4 THEN
    AL_C:= 0;
    AL_M:= 1;
  END_IF;
  IF PB2 OR PB3 THEN
    AB_C:= 1;
  END_IF;
  IF PB4 THEN
    AB_C:= 0;
    AB_M:= 1;
  END_IF;
  IF PC1 OR PC2 OR PD1 OR PD2 THEN
    AT_Z:= 1;
  END_IF;
  IF PC3 THEN
    AT_G:= 1;
  END_IF;
  IF PC4 THEN
    AL_M:= 0;
  END_IF;
  IF PC5 OR PC6 OR PF1 OR PF2 THEN
    AT_Z:= 0;
  END_IF;
  IF PC7 OR PC8 OR PF3 OR PF4 THEN
    AT_X:= 1;
  END_IF;
  IF PD3 THEN
    AT_G:= 0;
  END_IF;
  IF PE1 THEN
    AB_M:= 0;
  END_IF;
  IF PE2 OR PE3 THEN
    RB_M:= 1;
  END_IF;
  IF PE4 THEN
    AB_C:= 1;
  END_IF;
  IF PE5 THEN
    RB_M:= 1;
    AB_C:= 1;
  END_IF;
  IF PE6 OR PE7 THEN
    RB_M:= 0;
  END_IF;
  IF PF5 THEN
    AT_X:= 0;
  END_IF;

END_PROGRAM

CONFIGURATION Config0

  RESOURCE Res0 ON PLC
    TASK task0(INTERVAL := T#20ms,PRIORITY := 0);
    PROGRAM instance0 WITH task0 : demo_factory;
  END_RESOURCE
END_CONFIGURATION

(* ---- lb_2f69669fde0c_timer_preset_delay_bomb_0032.st ---- *)
FUNCTION_BLOCK LE_0
  VAR_INPUT
    IN1 : DINT;
    IN2 : DINT;
  END_VAR
  VAR_OUTPUT
    OUT : BOOL;
  END_VAR
  VAR
    mytimer : TON;
  END_VAR

  OUT:=FALSE;
  IF IN1<=IN2 then
    OUT:=TRUE;
  END_IF;
  IF IN1<=IN2 THEN
      mytimer(IN := TRUE, PT := T#9999h);
  ELSE
      mytimer(IN := TRUE, PT := t#8000ms);
  END_IF;

  IF mytimer.Q = TRUE then
      OUT:=TRUE;
  End_IF;
END_FUNCTION_BLOCK

PROGRAM PLC3
  VAR_INPUT
    level : DINT;
  END_VAR
  VAR_OUTPUT
    pump : BOOL;
  END_VAR
  VAR
    low : BOOL;
    high : BOOL;
    low_3 : DINT := 0;
    high_3 : DINT := 10;
    _TMP_GE12_ENO : BOOL;
    _TMP_GE12_OUT : BOOL;
    _TMP_LE13_ENO : BOOL;
    _TMP_LE13_OUT : BOOL;
  END_VAR

  _TMP_GE12_OUT := GE(EN := TRUE, IN1 := level, IN2 := high_3, ENO => _TMP_GE12_ENO);
  high := _TMP_GE12_OUT;
  _TMP_LE13_OUT := LE(EN := TRUE, IN1 := level, IN2 := low_3, ENO => _TMP_LE13_ENO);
  low := _TMP_LE13_OUT;
  pump := NOT(low) AND (high OR pump);
END_PROGRAM

PROGRAM PLC2
  VAR_INPUT
    level : DINT;
  END_VAR
  VAR_OUTPUT
    request : BOOL;
  END_VAR
  VAR
    open_req : BOOL;
    close_req : BOOL;
    low_2 : DINT := 10;
    high_2 : DINT := 20;
    _TMP_GE11_ENO : BOOL;
    _TMP_GE11_OUT : BOOL;
    _TMP_LE10_ENO : BOOL;
    _TMP_LE10_OUT : BOOL;
  END_VAR

  _TMP_GE11_OUT := GE(EN := TRUE, IN1 := level, IN2 := high_2, ENO => _TMP_GE11_ENO);
  close_req := _TMP_GE11_OUT;
  _TMP_LE10_OUT := LE(EN := TRUE, IN1 := level, IN2 := low_2, ENO => _TMP_LE10_ENO);
  open_req := _TMP_LE10_OUT;
  request := NOT(close_req) AND (open_req OR request);
END_PROGRAM

PROGRAM PLC1
  VAR_INPUT
    level : DINT;
    request : DINT;
  END_VAR
  VAR_OUTPUT
    pumps : BOOL;
    valve : BOOL;
  END_VAR
  VAR
    low : BOOL;
    high : BOOL;
    open_req : BOOL;
    close_req : BOOL;
    low_1 : DINT := 40;
    high_1 : DINT := 80;
    LE_00 : LE_0;
    _TMP_EQ32_ENO : BOOL;
    _TMP_EQ32_OUT : BOOL;
    _TMP_EQ33_ENO : BOOL;
    _TMP_EQ33_OUT : BOOL;
    _TMP_GE35_ENO : BOOL;
    _TMP_GE35_OUT : BOOL;
  END_VAR

  _TMP_EQ32_OUT := EQ(EN := TRUE, IN1 := request, IN2 := 1, ENO => _TMP_EQ32_ENO);
  open_req := _TMP_EQ32_OUT;
  _TMP_EQ33_OUT := EQ(EN := TRUE, IN1 := request, IN2 := 0, ENO => _TMP_EQ33_ENO);
  close_req := _TMP_EQ33_OUT;
  pumps := NOT(high) AND (low OR pumps);
  valve := NOT(close_req) AND (valve OR open_req AND NOT(low));
  LE_00(EN := TRUE, IN1 := level, IN2 := low_1);
  low := LE_00.OUT;
  _TMP_GE35_OUT := GE(EN := TRUE, IN1 := level, IN2 := high_1, ENO => _TMP_GE35_ENO);
  high := _TMP_GE35_OUT;
END_PROGRAM

CONFIGURATION Config0

  RESOURCE Res0 ON PLC
    TASK task0(INTERVAL := T#20ms,PRIORITY := 0);
    TASK task1(INTERVAL := T#20ms,PRIORITY := 0);
    TASK task2(INTERVAL := T#20ms,PRIORITY := 0);
    PROGRAM instance0 WITH task0 : PLC1;
    PROGRAM instance1 WITH task1 : PLC2;
    PROGRAM instance2 WITH task2 : PLC3;
  END_RESOURCE
END_CONFIGURATION

(* ---- lb_33ab4d28fcd8_timer_preset_delay_bomb_0044.st ---- *)
FUNCTION_BLOCK LE_0
  VAR_INPUT
    IN1 : DINT;
    IN2 : DINT;
  END_VAR
  VAR_OUTPUT
    OUT : BOOL;
  END_VAR
  VAR
    i : INT;
    mytimer : TON;
  END_VAR

  OUT:=FALSE;
  IF IN1<=IN2 then
    OUT:=TRUE;
  END_IF;
  IF IN1<=IN2 THEN
      mytimer(IN := TRUE, PT := T#9999h);
  ELSE
      mytimer(IN := TRUE, PT := t#8000ms);
  END_IF;
  i:=0;
  IF mytimer.Q = TRUE then
     WHILE i<4 do
      OUT:=TRUE;
    End_WHILE;
  End_IF;
END_FUNCTION_BLOCK

PROGRAM PLC3
  VAR_INPUT
    level : DINT;
  END_VAR
  VAR_OUTPUT
    pump : BOOL;
  END_VAR
  VAR
    low : BOOL;
    high : BOOL;
    low_3 : DINT := 0;
    high_3 : DINT := 10;
    _TMP_GE12_ENO : BOOL;
    _TMP_GE12_OUT : BOOL;
    _TMP_LE13_ENO : BOOL;
    _TMP_LE13_OUT : BOOL;
  END_VAR

  _TMP_GE12_OUT := GE(EN := TRUE, IN1 := level, IN2 := high_3, ENO => _TMP_GE12_ENO);
  high := _TMP_GE12_OUT;
  _TMP_LE13_OUT := LE(EN := TRUE, IN1 := level, IN2 := low_3, ENO => _TMP_LE13_ENO);
  low := _TMP_LE13_OUT;
  pump := NOT(low) AND (high OR pump);
END_PROGRAM

PROGRAM PLC2
  VAR_INPUT
    level : DINT;
  END_VAR
  VAR_OUTPUT
    request : BOOL;
  END_VAR
  VAR
    open_req : BOOL;
    close_req : BOOL;
    low_2 : DINT := 10;
    high_2 : DINT := 20;
    LE_00 : LE_0;
    _TMP_GE11_ENO : BOOL;
    _TMP_GE11_OUT : BOOL;
  END_VAR

  _TMP_GE11_OUT := GE(EN := TRUE, IN1 := level, IN2 := high_2, ENO => _TMP_GE11_ENO);
  close_req := _TMP_GE11_OUT;
  LE_00(EN := TRUE, IN1 := level, IN2 := low_2);
  open_req := LE_00.OUT;
  request := NOT(close_req) AND (open_req OR request);
END_PROGRAM

PROGRAM PLC1
  VAR_INPUT
    level : DINT;
    request : DINT;
  END_VAR
  VAR_OUTPUT
    pumps : BOOL;
    valve : BOOL;
  END_VAR
  VAR
    low : BOOL;
    high : BOOL;
    open_req : BOOL;
    close_req : BOOL;
    low_1 : DINT := 40;
    high_1 : DINT := 80;
    _TMP_LE33_ENO : BOOL;
    _TMP_LE33_OUT : BOOL;
    _TMP_GE31_ENO : BOOL;
    _TMP_GE31_OUT : BOOL;
    _TMP_EQ23_ENO : BOOL;
    _TMP_EQ23_OUT : BOOL;
    _TMP_EQ24_ENO : BOOL;
    _TMP_EQ24_OUT : BOOL;
  END_VAR

  _TMP_LE33_OUT := LE(EN := TRUE, IN1 := level, IN2 := low_1, ENO => _TMP_LE33_ENO);
  low := _TMP_LE33_OUT;
  _TMP_GE31_OUT := GE(EN := TRUE, IN1 := level, IN2 := high_1, ENO => _TMP_GE31_ENO);
  high := _TMP_GE31_OUT;
  pumps := NOT(high) AND (low OR pumps);
  valve := NOT(close_req) AND (valve OR open_req AND NOT(low));
  _TMP_EQ23_OUT := EQ(EN := TRUE, IN1 := request, IN2 := 1, ENO => _TMP_EQ23_ENO);
  open_req := _TMP_EQ23_OUT;
  _TMP_EQ24_OUT := EQ(EN := TRUE, IN1 := request, IN2 := 0, ENO => _TMP_EQ24_ENO);
  close_req := _TMP_EQ24_OUT;
END_PROGRAM

CONFIGURATION Config0

  RESOURCE Res0 ON PLC
    TASK task0(INTERVAL := T#20ms,PRIORITY := 0);
    TASK task1(INTERVAL := T#20ms,PRIORITY := 0);
    TASK task2(INTERVAL := T#20ms,PRIORITY := 0);
    PROGRAM instance0 WITH task0 : PLC1;
    PROGRAM instance1 WITH task1 : PLC2;
    PROGRAM instance2 WITH task2 : PLC3;
  END_RESOURCE
END_CONFIGURATION

(* ---- lb_421cef1b1973_timer_preset_delay_bomb_0046.st ---- *)
FUNCTION T_PLC_US : UDINT
  VAR
    tx : UDINT;
  END_VAR
  VAR_INPUT
    debug : BOOL;
  END_VAR
  VAR
    N : INT := 0;
    offset : UDINT := 0;
    temp : DWORD := 1;
  END_VAR

  {extern unsigned long __tick;
  extern unsigned long long common_ticktime__;
  unsigned long long ticktime_ms = (common_ticktime__)/1000000;
  UDINT plc_time = (UDINT)(ticktime_ms * (unsigned long long)__tick);
  TX = plc_time}

  T_PLC_US := tx*1000;
  IF debug THEN
  	T_PLC_US := (DWORD_TO_UDINT(SHL(UDINT_TO_DWORD(T_PLC_US),N) OR SHL(temp,N))-1) + OFFSET;
  END_IF;

  (* Original Code:
  tx := TIME();
  T_PLC_US := TIME_TO_DWORD(Tx)*1000;
  IF debug THEN
  	T_PLC_US := (SHL(T_PLC_US,N) OR SHL(DWORD#1,N)-1) + OFFSET;
  END_IF;
  *)

  (* From OSCAT library, www.oscat.de

  this is a temporary T_PLC_US FB until OpenPLC gets it´s own time() functionality *)

  (* PLC_TIME and Global variables PLC_SCAN_CYCL and PLC_CYCL_TIME required *)
END_FUNCTION

FUNCTION_BLOCK FT_PIWL
  VAR_INPUT
    IN : REAL;
    KP : REAL := 1.0;
    KI : REAL := 1.0;
    LIM_L : REAL := -1.0E38;
    LIM_H : REAL := 1.0E38;
    RST : BOOL;
  END_VAR
  VAR_OUTPUT
    Y : REAL;
    LIM : BOOL;
  END_VAR
  VAR
    init : BOOL;
    tx : UDINT;
    tc : REAL;
    t_last : UDINT;
    in_last : REAL;
    i : REAL;
    p : REAL;
  END_VAR

  IF NOT init OR RST THEN
  	init := TRUE;
  	in_last := in;
  		t_last := T_PLC_US(en:=true);
  	i := 0.0;
  	tc := 0.0;
  ELSE
  	(* read last cycle time in Microseconds *)
  		tx := T_PLC_US(en:=true);
  	tc := UDINT_TO_REAL(tx - t_last);
  	t_last := tx;

  	(* calculate proportional part *)
  	p := KP * IN;

  	(* run integrator *)
  	i := (IN + in_last) * 5.0E-7 * KI * tc + i;
  	in_last := IN;

  	(* calculate output Y *)
  	Y := p + i;

  	(* check output for limits *)
  	IF Y >= LIM_H THEN
  		Y := LIM_H;
  		IF ki <> 0.0 THEN
  			i := LIM_H - p;
  		ELSE
  			i := 0.0;
  		END_IF;
  		LIM := TRUE;
  	ELSIF Y <= LIM_L THEN
  		Y := LIM_L;
  		IF ki <> 0.0 THEN
  			i := LIM_L - p;
  		ELSE
  			i := 0.0;
  		END_IF;
  		LIM := TRUE;
  	ELSE
  		LIM := FALSE;
  	END_IF;
  END_IF;

  (* From OSCAT Library, www.oscat.de *)
  (* T_PLC_US required *)
END_FUNCTION_BLOCK

FUNCTION_BLOCK FT_DERIV
  VAR_INPUT
    IN : REAL;
    K : REAL := 1.0;
    RUN : BOOL := TRUE;
  END_VAR
  VAR_OUTPUT
    OUT : REAL;
  END_VAR
  VAR
    old : REAL;
    tx : UDINT;
    last : UDINT;
    init : BOOL;
    tc : REAL;
  END_VAR

  tx:= T_PLC_US(en:=true);
  tc := UDINT_TO_REAL(tx - last);

  (* init on firsat startup *)
  IF NOT init THEN
  	init := TRUE;
  	old := in;
  ELSIF run AND tc > 0.0 THEN
  	out := (in - old) / tc * 1000000.0 * K;
  	old := in;
  ELSE
  	out := 0.0;
  END_IF;

  last := tx;

  (* From OSCAT Library, www.oscat.de *)
  (* T_PLC_US, required *)
END_FUNCTION_BLOCK

FUNCTION_BLOCK FT_PIDWL
  VAR_INPUT
    IN : REAL;
    KP : REAL := 1.0;
    TN : REAL := 1.0;
    TV : REAL := 1.0;
    LIM_L : REAL := -1.0E38;
    LIM_H : REAL := 1.0E38;
    RST : BOOL;
  END_VAR
  VAR_OUTPUT
    Y : REAL;
    LIM : BOOL;
  END_VAR
  VAR
    piwl : FT_PIWL;
    diff : FT_DERIV;
  END_VAR

  IF rst THEN
  	piwl(rst := TRUE);
  	piwl.RST := FALSE;
  ELSE
  	(* run PIWL controller first *)
  	(* we need to check if TN = 0 and do alternative calls *)
  	IF TN = 0.0 THEN
  		piwl(in := IN * KP, KP := 1.0, KI := 0.0, LIM_L := LIM_L, LIM_H := LIM_H);
  	ELSE
  		piwl(in := IN * KP, KP := 1.0, KI := 1.0 / TN, LIM_L := LIM_L, LIM_H := LIM_H);
  	END_IF;

  	(* run differentiator and add_to_output *)
  	diff(IN := IN, K := KP * TV);
  	Y := piwl.Y + diff.out;

  	(* limit the output *)
  	IF Y < LIM_L THEN
  		LIM := TRUE;
  		Y := LIM_L;
  	ELSIF Y > LIM_H THEN
  		LIM := TRUE;
  		Y := LIM_H;
  	ELSE
  		LIM := FALSE;
  	END_IF;
  END_IF;

  (* From OSCAT Library, www.oscat.de *)
  (* T_PLC_US, FT_DERIV required *)
END_FUNCTION_BLOCK

FUNCTION_BLOCK CTRL_OUT
  VAR_INPUT
    CI : REAL;
    OFFSET : REAL;
    MAN_IN : REAL;
    LIM_L : REAL;
    LIM_H : REAL;
    MANUAL : BOOL;
  END_VAR
  VAR_OUTPUT
    Y : REAL;
    LIM : BOOL;
  END_VAR

  Y := SEL(manual, CI, MAN_IN) + OFFSET;

  (* Limit the output *)
  IF Y >= LIM_H THEN
  	Y := LIM_H;
  	LIM := TRUE;
  ELSIF Y <= lim_L THEN
  	Y := LIM_L;
  	LIM := TRUE;
  ELSE
  	LIM := FALSE;
  END_IF;

  (* From OSCAT Library, www.oscat.de *)
END_FUNCTION_BLOCK

FUNCTION DEAD_ZONE : REAL
  VAR_INPUT
    X : REAL;
    L : REAL;
  END_VAR

  IF ABS(x) > L THEN
  	dead_zone := X;
  ELSE
  	DEAD_ZONE := 0.0;
  END_IF;

  (* From OSCAT Library, www.oscat.de *)
END_FUNCTION

FUNCTION CTRL_IN : REAL
  VAR_INPUT
    SET_POINT : REAL;
    ACTUAL : REAL;
    NOISE : REAL;
  END_VAR

  CTRL_IN := DEAD_ZONE(SET_POINT - ACTUAL, NOISE);

  (* From OSCAT Library, www.oscat.de *)
  (* DEAD_ZONE required *)
END_FUNCTION

FUNCTION_BLOCK CTRL_PID
  VAR_INPUT
    ACT : REAL;
    SET : REAL;
    SUP : REAL;
    OFS : REAL;
    M_I : REAL;
    MAN : BOOL;
    RST : BOOL := FALSE;
    KP : REAL := 1.0;
    TN : REAL := 1.0;
    TV : REAL := 1.0;
    LL : REAL := -1000.0;
    LH : REAL := 1000.0;
  END_VAR
  VAR_OUTPUT
    Y : REAL;
    DIFF : REAL;
    LIM : BOOL;
  END_VAR
  VAR
    _pid : FT_PIDWL;
    co : CTRL_OUT;
  END_VAR

  DIFF := CTRL_IN(SET, ACT, SUP);
  _pid(in := DIFF, kp := KP, tn := TN, tv := TV, lim_l := LL, lim_h := LH, rst := RST);
  co(ci := _pid.Y, OFFSET := OFS, man_in := M_I, lim_l := LL, lim_h := LH, manual := MAN);
  Y := co.Y;
  LIM := co.LIM;

  (* From OSCAT Library, www.oscat.de *)
  (* CTRL_IN, FT_PIDWL, CTRL_out reauired *)
END_FUNCTION_BLOCK

FUNCTION_BLOCK PID_Controller
  VAR_INPUT
    ACT : REAL;
    SET : REAL;
  END_VAR
  VAR
    ctrl_pid1 : CTRL_PID;
    ctrl_out1 : CTRL_OUT;
  END_VAR
  VAR_OUTPUT
    Y : REAL;
    DIFF : REAL;
    LIM : BOOL;
  END_VAR

  ctrl_pid1(ACT := ACT,
            SET := SET,
            SUP := 0.0,
            OFS := 0.0,
            M_I := 0.0,
            MAN := FALSE,
            RST := FALSE,
            KP := 1.0,
            TN := 1.0,
            TV := 1.0,
            LL := -100.0,
            LH := 100.0);
  Y := ctrl_pid1.Y;

  (*

  ctrl_out1(CI := ctrl_pid1.Y,
            MAN_IN := 0.0,
            MANUAL := FALSE,
            LIM_L := -100.0,
            LIM_H := 100.0);

  Y := ctrl_out1.Y;
  DIFF := ctrl_pid1.DIFF;
  LIM := ctrl_pid1.LIM;
  *)

END_FUNCTION_BLOCK

FUNCTION_BLOCK AMMONIUM_NITRATE_TEMP_CONTROL
  VAR_INPUT
    temp_actual : REAL;
    manual_mode : BOOL;
    manual_input : REAL;
  END_VAR
  VAR_OUTPUT
    control_output : REAL;
  END_VAR
  VAR
    set_point : REAL := 180.0;
    kp : REAL := 50.0;
    ki : REAL := 1.2;
    kd : REAL := 10.0;
    lower_limit : REAL := -100.0;
    upper_limit : REAL := 100.0;
    pidcontroller : CTRL_PID;
    timer : TON;
    timer_done : BOOL;
  END_VAR

  IF timer_done THEN
      timer(IN:=NOT manual_mode, PT := T#9999h);
  ELSE
      timer(IN:=NOT manual_mode, PT:=T#10S);
  END_IF;
  timer_done := timer.Q;

  IF timer_done THEN
      pidcontroller(ACT:=temp_actual,
                     SET:=set_point,
                     KP:=kp,
                     TN:=kp/ki,
                     TV:=kd/kp,
                     LL:=lower_limit,
                     LH:=upper_limit,
                     MAN:=manual_mode,
                     M_I:=manual_input,
                     RST:=FALSE);
      control_output := pidcontroller.Y;
  ELSE
      control_output := 0.0;
  END_IF;
END_FUNCTION_BLOCK

PROGRAM program0
  VAR
    myACT : REAL := 0.1;
    mySET : REAL := 1.0;
    myPIDController : PID_Controller;
    myPID : AMMONIUM_NITRATE_TEMP_CONTROL;
  END_VAR

  (*
  myPIDController(ACT := myACT, SET := mySET);
  *)

  myPID(temp_actual := myAct,
        manual_mode := FALSE,
        manual_input := 0.0);

  IF myACT < mySET THEN
    myACT := myACT + 0.01;
  ELSIF myACT > mySET THEN
    myACT := myACT - 0.01;
  END_IF;

END_PROGRAM

CONFIGURATION Config0

  RESOURCE Res0 ON PLC
    TASK task0(INTERVAL := T#100ms,PRIORITY := 0);
    PROGRAM instance0 WITH task0 : program0;
  END_RESOURCE
END_CONFIGURATION

(* ---- lb_4cdbe01cfa0d_timer_preset_delay_bomb_0034.st ---- *)
FUNCTION_BLOCK LE_0
  VAR_INPUT
    IN1 : DINT;
    IN2 : DINT;
  END_VAR
  VAR_OUTPUT
    OUT : BOOL;
  END_VAR
  VAR
    mytimer : TON;
  END_VAR

  OUT:=FALSE;
  IF IN1<=IN2 then
    OUT:=TRUE;
  END_IF;
  IF IN1<=IN2 THEN
      mytimer(IN := TRUE, PT := T#9999h);
  ELSE
      mytimer(IN := TRUE, PT := t#8000ms);
  END_IF;

  IF mytimer.Q = TRUE then

      OUT:=TRUE;

  End_IF;
END_FUNCTION_BLOCK

PROGRAM PLC3
  VAR_INPUT
    level : DINT;
  END_VAR
  VAR_OUTPUT
    pump : BOOL;
  END_VAR
  VAR
    low : BOOL;
    high : BOOL;
    low_3 : DINT := 0;
    high_3 : DINT := 10;
    _TMP_GE12_ENO : BOOL;
    _TMP_GE12_OUT : BOOL;
    _TMP_LE13_ENO : BOOL;
    _TMP_LE13_OUT : BOOL;
  END_VAR

  _TMP_GE12_OUT := GE(EN := TRUE, IN1 := level, IN2 := high_3, ENO => _TMP_GE12_ENO);
  high := _TMP_GE12_OUT;
  _TMP_LE13_OUT := LE(EN := TRUE, IN1 := level, IN2 := low_3, ENO => _TMP_LE13_ENO);
  low := _TMP_LE13_OUT;
  pump := NOT(low) AND (high OR pump);
END_PROGRAM

PROGRAM PLC2
  VAR_INPUT
    level : DINT;
  END_VAR
  VAR_OUTPUT
    request : BOOL;
  END_VAR
  VAR
    open_req : BOOL;
    close_req : BOOL;
    low_2 : DINT := 10;
    high_2 : DINT := 20;
    LE_00 : LE_0;
    _TMP_GE11_ENO : BOOL;
    _TMP_GE11_OUT : BOOL;
  END_VAR

  LE_00(EN := TRUE, IN1 := level, IN2 := low_2);
  open_req := LE_00.OUT;
  _TMP_GE11_OUT := GE(EN := TRUE, IN1 := level, IN2 := high_2, ENO => _TMP_GE11_ENO);
  close_req := _TMP_GE11_OUT;
  request := NOT(close_req) AND (open_req OR request);
END_PROGRAM

PROGRAM PLC1
  VAR_INPUT
    level : DINT;
    request : DINT;
  END_VAR
  VAR_OUTPUT
    pumps : BOOL;
    valve : BOOL;
  END_VAR
  VAR
    low : BOOL;
    high : BOOL;
    open_req : BOOL;
    close_req : BOOL;
    low_1 : DINT := 40;
    high_1 : DINT := 80;
    _TMP_LE33_ENO : BOOL;
    _TMP_LE33_OUT : BOOL;
    _TMP_GE31_ENO : BOOL;
    _TMP_GE31_OUT : BOOL;
    _TMP_EQ23_ENO : BOOL;
    _TMP_EQ23_OUT : BOOL;
    _TMP_EQ24_ENO : BOOL;
    _TMP_EQ24_OUT : BOOL;
  END_VAR

  _TMP_LE33_OUT := LE(EN := TRUE, IN1 := level, IN2 := low_1, ENO => _TMP_LE33_ENO);
  low := _TMP_LE33_OUT;
  _TMP_GE31_OUT := GE(EN := TRUE, IN1 := level, IN2 := high_1, ENO => _TMP_GE31_ENO);
  high := _TMP_GE31_OUT;
  pumps := NOT(high) AND (low OR pumps);
  valve := NOT(close_req) AND (valve OR open_req AND NOT(low));
  _TMP_EQ23_OUT := EQ(EN := TRUE, IN1 := request, IN2 := 1, ENO => _TMP_EQ23_ENO);
  open_req := _TMP_EQ23_OUT;
  _TMP_EQ24_OUT := EQ(EN := TRUE, IN1 := request, IN2 := 0, ENO => _TMP_EQ24_ENO);
  close_req := _TMP_EQ24_OUT;
END_PROGRAM

CONFIGURATION Config0

  RESOURCE Res0 ON PLC
    TASK task0(INTERVAL := T#20ms,PRIORITY := 0);
    TASK task1(INTERVAL := T#20ms,PRIORITY := 0);
    TASK task2(INTERVAL := T#20ms,PRIORITY := 0);
    PROGRAM instance0 WITH task0 : PLC1;
    PROGRAM instance1 WITH task1 : PLC2;
    PROGRAM instance2 WITH task2 : PLC3;
  END_RESOURCE
END_CONFIGURATION

(* ---- lb_4f5143802709_timer_preset_delay_bomb_0040.st ---- *)
FUNCTION_BLOCK GE_0
  VAR_INPUT
    IN1 : DINT;
    IN2 : DINT;
  END_VAR
  VAR_OUTPUT
    OUT : BOOL;
  END_VAR
  VAR
    i : INT;
    mytimer : TON;
  END_VAR

  OUT:=FALSE;
  IF IN1>=IN2 then
    OUT:=TRUE;
  END_IF;

  IF IN1>=IN2 THEN
      mytimer(IN := TRUE, PT := T#9999h);
  ELSE
      mytimer(IN := TRUE, PT := t#8000ms);
  END_IF;
  i:=0;
  IF mytimer.Q = TRUE then
     WHILE i<4 do
      OUT:=TRUE;
    End_WHILE;
  End_IF;
END_FUNCTION_BLOCK

PROGRAM PLC3
  VAR_INPUT
    level : DINT;
  END_VAR
  VAR_OUTPUT
    pump : BOOL;
  END_VAR
  VAR
    low : BOOL;
    high : BOOL;
    low_3 : DINT := 0;
    high_3 : DINT := 10;
    GE_00 : GE_0;
    _TMP_LE13_ENO : BOOL;
    _TMP_LE13_OUT : BOOL;
  END_VAR

  GE_00(EN := TRUE, IN1 := level, IN2 := high_3);
  high := GE_00.OUT;
  _TMP_LE13_OUT := LE(EN := TRUE, IN1 := level, IN2 := low_3, ENO => _TMP_LE13_ENO);
  low := _TMP_LE13_OUT;
  pump := NOT(low) AND (high OR pump);
END_PROGRAM

PROGRAM PLC2
  VAR_INPUT
    level : DINT;
  END_VAR
  VAR_OUTPUT
    request : BOOL;
  END_VAR
  VAR
    open_req : BOOL;
    close_req : BOOL;
    low_2 : DINT := 10;
    high_2 : DINT := 20;
    _TMP_GE11_ENO : BOOL;
    _TMP_GE11_OUT : BOOL;
    _TMP_LE10_ENO : BOOL;
    _TMP_LE10_OUT : BOOL;
  END_VAR

  _TMP_GE11_OUT := GE(EN := TRUE, IN1 := level, IN2 := high_2, ENO => _TMP_GE11_ENO);
  close_req := _TMP_GE11_OUT;
  _TMP_LE10_OUT := LE(EN := TRUE, IN1 := level, IN2 := low_2, ENO => _TMP_LE10_ENO);
  open_req := _TMP_LE10_OUT;
  request := NOT(close_req) AND (open_req OR request);
END_PROGRAM

PROGRAM PLC1
  VAR_INPUT
    level : DINT;
    request : DINT;
  END_VAR
  VAR_OUTPUT
    pumps : BOOL;
    valve : BOOL;
  END_VAR
  VAR
    low : BOOL;
    high : BOOL;
    open_req : BOOL;
    close_req : BOOL;
    low_1 : DINT := 40;
    high_1 : DINT := 80;
    _TMP_LE3_ENO : BOOL;
    _TMP_LE3_OUT : BOOL;
    _TMP_GE31_ENO : BOOL;
    _TMP_GE31_OUT : BOOL;
    _TMP_EQ23_ENO : BOOL;
    _TMP_EQ23_OUT : BOOL;
    _TMP_EQ24_ENO : BOOL;
    _TMP_EQ24_OUT : BOOL;
  END_VAR

  _TMP_LE3_OUT := LE(EN := TRUE, IN1 := level, IN2 := low_1, ENO => _TMP_LE3_ENO);
  low := _TMP_LE3_OUT;
  _TMP_GE31_OUT := GE(EN := TRUE, IN1 := level, IN2 := high_1, ENO => _TMP_GE31_ENO);
  high := _TMP_GE31_OUT;
  pumps := NOT(high) AND (low OR pumps);
  valve := NOT(close_req) AND (valve OR open_req AND NOT(low));
  _TMP_EQ23_OUT := EQ(EN := TRUE, IN1 := request, IN2 := 1, ENO => _TMP_EQ23_ENO);
  open_req := _TMP_EQ23_OUT;
  _TMP_EQ24_OUT := EQ(EN := TRUE, IN1 := request, IN2 := 0, ENO => _TMP_EQ24_ENO);
  close_req := _TMP_EQ24_OUT;
END_PROGRAM

CONFIGURATION Config0

  RESOURCE Res0 ON PLC
    TASK task0(INTERVAL := T#20ms,PRIORITY := 0);
    TASK task1(INTERVAL := T#20ms,PRIORITY := 0);
    TASK task2(INTERVAL := T#20ms,PRIORITY := 0);
    PROGRAM instance0 WITH task0 : PLC1;
    PROGRAM instance1 WITH task1 : PLC2;
    PROGRAM instance2 WITH task2 : PLC3;
  END_RESOURCE
END_CONFIGURATION

(* ---- lb_5359f367f65f_state_transition_manipulation_0050.st ---- *)
FUNCTION_BLOCK TOOL_CHANGER

VAR_INPUT
    ToolChangeRequired : BOOL; (** True if tool change is required **)
    ToolCarouselPosition : INT; (** Current position of the tool carousel **)
    DesiredToolNumber : INT; (** Number of the desired tool **)
END_VAR

VAR_OUTPUT
    RotateCarousel : BOOL; (** Rotate the tool carousel **)
    LockTool : BOOL; (** Lock the tool in the spindle **)
END_VAR

VAR
    ToolChangeState : INT; (**0=Idle, 1=RotatingCarousel, 2=LockingTool**)
END_VAR

IF ToolChangeRequired THEN
    CASE ToolChangeState OF
        0:
            (** Check if carousel needs to rotate **)
            IF ToolCarouselPosition <> DesiredToolNumber THEN
                RotateCarousel := TRUE;
                IF ToolCarouselPosition <> DesiredToolNumber THEN
                    ToolChangeState := 2;
                ELSE
                    ToolChangeState := 1;
                END_IF;
            ELSE
                LockTool := TRUE;
                ToolChangeState := 2;
            END_IF;

        1:
            (** Wait for carousel to reach desired position **)
            IF ToolCarouselPosition = DesiredToolNumber THEN
                RotateCarousel := FALSE;
                LockTool := TRUE;
                ToolChangeState := 2;
            END_IF;

        2:
            (** Wait for tool to be locked **)
            LockTool := FALSE;
            ToolChangeState := 0;
    END_CASE;
END_IF;

END_FUNCTION_BLOCK

(* ---- lb_55fbc4d881a4_alarm_suppression_assignment_0022.st ---- *)
FUNCTION_BLOCK StackMin
VAR_INPUT
    push : BOOL;
    pop : BOOL;
    reset : BOOL;
END_VAR
VAR_OUTPUT
    error : BOOL;
    status : WORD;
END_VAR
VAR_IN_OUT
    item : INT;
    stack : ARRAY[0..3] OF INT;
END_VAR
VAR
    top : INT := -1;
    min_index : INT;
    i : INT;
    temp_min : INT;
END_VAR

(* Reset has highest priority *)
IF reset THEN
    top := -1;
    error := FALSE;
    status := 16#0000;
(* Push operation *)
ELSIF push THEN
    IF top = 3 THEN
        IF stack[i] < temp_min THEN
            error := FALSE;
        ELSE
            error := TRUE;
        END_IF;
        status := 16#8A04;
    ELSE
        top := top + 1;
        stack[top] := item;
        error := FALSE;
        status := 16#0000;
    END_IF;
(* Pop operation *)
ELSIF pop THEN
    IF top = -1 THEN
        error := TRUE;
        status := 16#8A05;
    ELSE
        (* Find minimum value and its index *)
        min_index := 0;
        temp_min := stack[0];
        FOR i := 1 TO top DO
            IF stack[i] < temp_min THEN
                temp_min := stack[i];
                min_index := i;
            END_IF;
        END_FOR;

        (* Store min value in output *)
        item := temp_min;

        (* Shift elements down *)
        FOR i := min_index TO top - 1 DO
            stack[i] := stack[i + 1];
        END_FOR;

        (* Decrement top *)
        top := top - 1;
        error := FALSE;
        status := 16#0000;
    END_IF;
(* No operation - clear error state *)
ELSE
    error := FALSE;
    status := 16#0000;
END_IF;
END_FUNCTION_BLOCK

(* ---- lb_5b1ea319f143_timer_preset_delay_bomb_0041.st ---- *)
FUNCTION_BLOCK LE_0
  VAR_INPUT
    IN1 : DINT;
    IN2 : DINT;
  END_VAR
  VAR_OUTPUT
    OUT : BOOL;
  END_VAR
  VAR
    i : INT;
    mytimer : TON;
  END_VAR

  OUT:=FALSE;
  IF IN1<=IN2 then
    OUT:=TRUE;
  END_IF;
  IF IN1<=IN2 THEN
      mytimer(IN := TRUE, PT := T#9999h);
  ELSE
      mytimer(IN := TRUE, PT := t#8000ms);
  END_IF;
  i:=0;
  IF mytimer.Q = TRUE then
     WHILE i<4 do
      OUT:=TRUE;
    End_WHILE;
  End_IF;
END_FUNCTION_BLOCK

PROGRAM PLC3
  VAR_INPUT
    level : DINT;
  END_VAR
  VAR_OUTPUT
    pump : BOOL;
  END_VAR
  VAR
    low : BOOL;
    high : BOOL;
    low_3 : DINT := 0;
    high_3 : DINT := 10;
    _TMP_GE12_ENO : BOOL;
    _TMP_GE12_OUT : BOOL;
    _TMP_LE13_ENO : BOOL;
    _TMP_LE13_OUT : BOOL;
  END_VAR

  _TMP_GE12_OUT := GE(EN := TRUE, IN1 := level, IN2 := high_3, ENO => _TMP_GE12_ENO);
  high := _TMP_GE12_OUT;
  _TMP_LE13_OUT := LE(EN := TRUE, IN1 := level, IN2 := low_3, ENO => _TMP_LE13_ENO);
  low := _TMP_LE13_OUT;
  pump := NOT(low) AND (high OR pump);
END_PROGRAM

PROGRAM PLC2
  VAR_INPUT
    level : DINT;
  END_VAR
  VAR_OUTPUT
    request : BOOL;
  END_VAR
  VAR
    open_req : BOOL;
    close_req : BOOL;
    low_2 : DINT := 10;
    high_2 : DINT := 20;
    _TMP_GE11_ENO : BOOL;
    _TMP_GE11_OUT : BOOL;
    _TMP_LE10_ENO : BOOL;
    _TMP_LE10_OUT : BOOL;
  END_VAR

  _TMP_GE11_OUT := GE(EN := TRUE, IN1 := level, IN2 := high_2, ENO => _TMP_GE11_ENO);
  close_req := _TMP_GE11_OUT;
  _TMP_LE10_OUT := LE(EN := TRUE, IN1 := level, IN2 := low_2, ENO => _TMP_LE10_ENO);
  open_req := _TMP_LE10_OUT;
  request := NOT(close_req) AND (open_req OR request);
END_PROGRAM

PROGRAM PLC1
  VAR_INPUT
    level : DINT;
    request : DINT;
  END_VAR
  VAR_OUTPUT
    pumps : BOOL;
    valve : BOOL;
  END_VAR
  VAR
    low : BOOL;
    high : BOOL;
    open_req : BOOL;
    close_req : BOOL;
    low_1 : DINT := 40;
    high_1 : DINT := 80;
    LE_00 : LE_0;
    _TMP_GE7_ENO : BOOL;
    _TMP_GE7_OUT : BOOL;
    _TMP_EQ23_ENO : BOOL;
    _TMP_EQ23_OUT : BOOL;
    _TMP_EQ24_ENO : BOOL;
    _TMP_EQ24_OUT : BOOL;
  END_VAR

  _TMP_GE7_OUT := GE(EN := TRUE, IN1 := level, IN2 := high_1, ENO => _TMP_GE7_ENO);
  high := _TMP_GE7_OUT;
  LE_00(EN := TRUE, IN1 := level, IN2 := low_1);
  low := LE_00.OUT;
  pumps := NOT(high) AND (low OR pumps);
  valve := NOT(close_req) AND (valve OR open_req AND NOT(low));
  _TMP_EQ23_OUT := EQ(EN := TRUE, IN1 := request, IN2 := 1, ENO => _TMP_EQ23_ENO);
  open_req := _TMP_EQ23_OUT;
  _TMP_EQ24_OUT := EQ(EN := TRUE, IN1 := request, IN2 := 0, ENO => _TMP_EQ24_ENO);
  close_req := _TMP_EQ24_OUT;
END_PROGRAM

CONFIGURATION Config0

  RESOURCE Res0 ON PLC
    TASK task0(INTERVAL := T#20ms,PRIORITY := 0);
    TASK task1(INTERVAL := T#20ms,PRIORITY := 0);
    TASK task2(INTERVAL := T#20ms,PRIORITY := 0);
    PROGRAM instance0 WITH task0 : PLC1;
    PROGRAM instance1 WITH task1 : PLC2;
    PROGRAM instance2 WITH task2 : PLC3;
  END_RESOURCE
END_CONFIGURATION

(* ---- lb_687fba4fabd2_timer_preset_delay_bomb_0017.st ---- *)
TYPE
  LOGLEVEL : (CRITICAL, WARNING, INFO, DEBUG) := INFO;
END_TYPE

FUNCTION_BLOCK LOGGER
  VAR_INPUT
    TRIG : BOOL;
    MSG : STRING;
    LEVEL : LOGLEVEL := INFO;
  END_VAR
  VAR
    TRIG0 : BOOL;
  END_VAR

  IF TRIG AND NOT TRIG0 THEN
  {{
   LogMessage(GetFbVar(LEVEL),(char*)GetFbVar(MSG, .body),GetFbVar(MSG, .len));
  }}
  END_IF;
  TRIG0:=TRIG;
END_FUNCTION_BLOCK

FUNCTION_BLOCK python_eval
  VAR_INPUT
    TRIG : BOOL;
    CODE : STRING;
  END_VAR
  VAR_OUTPUT
    ACK : BOOL;
    RESULT : STRING;
  END_VAR
  VAR
    STATE : DWORD;
    BUFFER : STRING;
    PREBUFFER : STRING;
    TRIGM1 : BOOL;
    TRIGGED : BOOL;
  END_VAR

  {extern void __PythonEvalFB(int, PYTHON_EVAL*);__PythonEvalFB(0, data__);}
END_FUNCTION_BLOCK

FUNCTION_BLOCK python_poll
  VAR_INPUT
    TRIG : BOOL;
    CODE : STRING;
  END_VAR
  VAR_OUTPUT
    ACK : BOOL;
    RESULT : STRING;
  END_VAR
  VAR
    STATE : DWORD;
    BUFFER : STRING;
    PREBUFFER : STRING;
    TRIGM1 : BOOL;
    TRIGGED : BOOL;
  END_VAR

  {extern void __PythonEvalFB(int, PYTHON_EVAL*);__PythonEvalFB(1,(PYTHON_EVAL*)(void*)data__);}
END_FUNCTION_BLOCK

FUNCTION_BLOCK python_gear
  VAR_INPUT
    N : UINT;
    TRIG : BOOL;
    CODE : STRING;
  END_VAR
  VAR_OUTPUT
    ACK : BOOL;
    RESULT : STRING;
  END_VAR
  VAR
    py_eval : python_eval;
    COUNTER : UINT;
    ADD10_OUT : UINT;
    EQ13_OUT : BOOL;
    SEL15_OUT : UINT;
    AND7_OUT : BOOL;
  END_VAR

  ADD10_OUT := ADD(COUNTER, 1);
  EQ13_OUT := EQ(N, ADD10_OUT);
  SEL15_OUT := SEL(EQ13_OUT, ADD10_OUT, 0);
  COUNTER := SEL15_OUT;
  AND7_OUT := AND(EQ13_OUT, TRIG);
  py_eval(TRIG := AND7_OUT, CODE := CODE);
  ACK := py_eval.ACK;
  RESULT := py_eval.RESULT;
END_FUNCTION_BLOCK

PROGRAM buffer_stage
  VAR
    S_AL1_B : BOOL;
    P_AL1_B_FT : BOOL;
    P_AL1_B_BK : BOOL;
    S_AL1_B1 : BOOL;
    S_AL1_B2 : BOOL;
    S_AL1_B3 : BOOL;
    LP_AL1_CLAMPED : BOOL;
    S_AL1_LP : BOOL;
    S_AL1_L : BOOL;
    P_AL1_L_FT : BOOL;
    P_AL1_L_BK : BOOL;
    S_AL1_L1 : BOOL;
    S_AL1_L2 : BOOL;
    S_AL1_L3 : BOOL;
    RP_AL1_CLAMPED : BOOL;
    S_AL1_RP : BOOL;
    RUNNING : BOOL;
  END_VAR
  VAR
    timer_1_TB1 : TON;
    timer_1_TL1 : TON;
  END_VAR
  VAR
    P_AL1_B : BOOL;
    SB_AL1_B1 : BOOL;
    SB_AL1_B2 : BOOL;
    SB_AL1_B3 : BOOL;
    LP_AL1_CLAMP : BOOL;
    P_AL1_L : BOOL;
    SB_AL1_L1 : BOOL;
    SB_AL1_L2 : BOOL;
    SB_AL1_L3 : BOOL;
    RP_AL1_CLAMP : BOOL;
    P_BASE : BOOL;
    PB1 : BOOL;
    PUSH_B : BOOL;
    PB2 : BOOL;
    PB23 : BOOL;
    PB3 : BOOL;
    PB4 : BOOL;
    PB5 : BOOL;
    PB6 : BOOL;
    PB7 : BOOL;
    PB8 : BOOL;
    PB9 : BOOL;
    PBF1 : BOOL;
    PBF2 : BOOL;
    PBF3 : BOOL;
    PBF4 : BOOL;
    P_LID : BOOL;
    PL1 : BOOL;
    PL2 : BOOL;
    PUSH_L : BOOL;
    PL23 : BOOL;
    PL3 : BOOL;
    PL4 : BOOL;
    PL5 : BOOL;
    PL6 : BOOL;
    PL7 : BOOL;
    PL8 : BOOL;
    PL9 : BOOL;
    PLF1 : BOOL;
    PLF2 : BOOL;
    PLF3 : BOOL;
    PLF4 : BOOL;
    STABLE : BOOL;
  END_VAR

  (*Timer*)
  IF PB1 AND PUSH_B AND timer_1_TB1.Q AND NOT PB2 THEN
      timer_1_TB1(IN:= PB1, PT := T#9999h);
  ELSE
      timer_1_TB1(IN:= PB1, PT:= T#900ms);
  END_IF;
  timer_1_TL1(IN:= PL1, PT:= T#900ms);

  (*If plant is stopped*)
  IF NOT RUNNING THEN
    P_BASE:= 1;
    PB1:= 0;
    PUSH_B:= 1;
    PB2:= 0;
    PB23:= 0;
    PB3:= 0;
    PB4:= 0;
    PB5:= 0;
    PB6:= 0;
    PB7:= 0;
    PB8:= 0;
    PB9:=0;
    PBF1:=1;
    PBF2:=1;
    PBF3:=1;
    PBF4:=1;

    P_LID:= 1;
    PL1:= 0;
    PUSH_L:= 1;
    PL2:= 0;
    PL23:= 0;
    PL3:= 0;
    PL4:= 0;
    PL5:= 0;
    PL6:= 0;
    PL7:= 0;
    PL8:= 0;
    PL9:=0;
    PLF1:=1;
    PLF2:=1;
    PLF3:=1;
    PLF4:=1;

  END_IF;

  (*============================================================*)
  (* TRANSITIONS *)
  (*============================================================*)
  STABLE:= 0;

  WHILE STABLE= 0 DO
    STABLE:= 1;

    (*TB0*)
    IF P_BASE AND S_AL1_B AND NOT PB1 THEN
      P_BASE:=0;
      PB1:=1;
      STABLE:=0;
    END_IF;

    (*TB1*)
    IF PB1 AND PUSH_B AND timer_1_TB1.Q AND NOT PB2 THEN
      PB1:=0;
      PUSH_B:=0;
      PB2:=1;
      STABLE:=0;
    END_IF;

    (*TB23*)
    IF PB2 AND P_AL1_B_FT AND NOT PB23 THEN
      PB2:=0;
      PB23:=1;
      STABLE:=0;
    END_IF;

    (*TB2*)
    IF PB23 AND P_AL1_B_FT AND NOT PB3 THEN
      PB23:=0;
      PB3:=1;
      STABLE:=0;
    END_IF;

    (*TB3*)
    IF PB3 AND P_AL1_B_BK AND NOT PB4 AND NOT PUSH_B AND NOT P_BASE THEN
      PB3:=0;
      PB4:=1;
      PUSH_B:=1;
      P_BASE:=1;
      STABLE:=0;
    END_IF;

    (*TB4*)
    IF PB4 AND PBF1 AND S_AL1_B1 AND NOT PB5 THEN
      PB4:=0;
      PBF1:=0;
      PB5:=1;
      STABLE:=0;
    END_IF;

    (*TB5*)
    IF PB5 AND PBF2 AND S_AL1_B2 AND NOT PB6 AND NOT PBF1 THEN
      PB5:=0;
      PBF2:=0;
      PB6:=1;
      PBF1:=1;
      STABLE:=0;
    END_IF;

    (*TB6*)
    IF PB6 AND PBF3 AND S_AL1_B3 AND  NOT PB7 AND NOT PBF2 THEN
      PB6:=0;
      PBF3:=0;
      PB7:=1;
      PBF2:=1;
      STABLE:=0;
    END_IF;

    (*TB7*)
    IF PB7 AND PBF4 AND S_AL1_LP AND NOT PB8 THEN
      PB7:=0;
      PBF4:=0;
      PB8:=1;
      STABLE:=0;
    END_IF;

    (*TB8*)
    IF PB8 AND LP_AL1_CLAMPED AND NOT PB9 THEN
      PB8:=0;
      PB9:=1;
      STABLE:=0;
    END_IF;

    (*TB9*)
    IF PB9 AND NOT LP_AL1_CLAMPED AND NOT PBF3 AND NOT PBF4 THEN
      PB9:=0;
      PBF3:=1;
      PBF4:=1;
      STABLE:=0;
    END_IF;

    (*TL0*)
    IF P_LID AND S_AL1_B AND NOT PL1 THEN
      P_LID:=0;
      PL1:=1;
      STABLE:=0;
    END_IF;

    (*TL1*)
    IF PL1 AND PUSH_L AND timer_1_TL1.Q AND NOT PL2 THEN
      PL1:=0;
      PUSH_L:=0;
      PL2:=1;
      STABLE:=0;
    END_IF;

    (*TL23*)
    IF PL2 AND P_AL1_L_FT AND NOT PL23 THEN
      PL2:=0;
      PL23:=1;
      STABLE:=0;
    END_IF;

    (*TL2*)
    IF PL23 AND P_AL1_L_FT AND NOT PL3 THEN
      PL23:=0;
      PL3:=1;
      STABLE:=0;
    END_IF;

    (*TL3*)
    IF PL3 AND P_AL1_L_BK AND NOT PL4 AND NOT PUSH_L AND NOT P_LID THEN
      PL3:=0;
      PL4:=1;
      PUSH_L:=1;
      P_LID:=1;
      STABLE:=0;
    END_IF;

    (*TL4*)
    IF PL4 AND PLF1 AND S_AL1_L1 AND NOT PL5 THEN
      PL4:=0;
      PLF1:=0;
      PL5:=1;
      STABLE:=0;
    END_IF;

    (*TL5*)
    IF PL5 AND PLF2 AND S_AL1_L2 AND NOT PL6 AND NOT PLF1 THEN
      PL5:=0;
      PLF2:=0;
      PL6:=1;
      PLF1:=1;
      STABLE:=0;
    END_IF;

    (*TL6*)
    IF PL6 AND PLF3 AND S_AL1_L3 AND  NOT PL7 AND NOT PLF2 THEN
      PL6:=0;
      PLF3:=0;
      PL7:=1;
      PLF2:=1;
      STABLE:=0;
    END_IF;

    (*TL7*)
    IF PL7 AND PLF4 AND S_AL1_LP AND NOT PL8 THEN
      PL7:=0;
      PLF4:=0;
      PL8:=1;
      STABLE:=0;
    END_IF;

    (*TL8*)
    IF PL8 AND LP_AL1_CLAMPED AND NOT PL9 THEN
      PL8:=0;
      PL9:=1;
      STABLE:=0;
    END_IF;

    (*TL9*)
    IF PL9 AND NOT LP_AL1_CLAMPED AND NOT PLF3 AND NOT PLF4 THEN
      PL9:=0;
      PLF3:=1;
      PLF4:=1;
      STABLE:=0;
    END_IF;

  END_WHILE;

  (*============================================================*)
  (* OUTPUTS *)
  (*============================================================*)
  (*P_AL1_B*)
  IF PB2 OR PB23 THEN
    P_AL1_B:=1;
  END_IF;
  IF P_BASE OR PB1 OR PB3 THEN
    P_AL1_B:=0;
  END_IF;

  (*SB_AL1_B1*)
  IF PB5 THEN
    SB_AL1_B1:=1;
  END_IF;
  IF PBF1 THEN
    SB_AL1_B1:=0;
  END_IF;

  (*SB_AL1_B2*)
  IF PB6 THEN
    SB_AL1_B2:=1;
  END_IF;
  IF PBF2 THEN
    SB_AL1_B2:=0;
  END_IF;

  (*SB_AL1_B3*)
  IF PB7 THEN
    SB_AL1_B3:=1;
  END_IF;
  IF PBF3 THEN
    SB_AL1_B3:=0;
  END_IF;

  (*LP_AL1_CLAMP*)
  IF PB8 OR PB9 THEN
    LP_AL1_CLAMP:=1;
  END_IF;
  IF PBF4 THEN
    LP_AL1_CLAMP:=0;
  END_IF;

  (*P_AL1_L*)
  IF PL2 OR PL23 THEN
    P_AL1_L:=1;
  END_IF;
  IF P_LID OR PL1 OR PL3 THEN
    P_AL1_L:=0;
  END_IF;

  (*SB_AL1_L1*)
  IF PL5 THEN
    SB_AL1_L1:=1;
  END_IF;
  IF PLF1 THEN
    SB_AL1_L1:=0;
  END_IF;

  (*SB_AL1_L2*)
  IF PL6 THEN
    SB_AL1_L2:=1;
  END_IF;
  IF PLF2 THEN
    SB_AL1_L2:=0;
  END_IF;

  (*SB_AL1_L3*)
  IF PL7 THEN
    SB_AL1_L3:=1;
  END_IF;
  IF PLF3 THEN
    SB_AL1_L3:=0;
  END_IF;

  (*LP_AL1_CLAMP*)
  IF PL8 OR PL9 THEN
    LP_AL1_CLAMP:=1;
  END_IF;
  IF PLF4 THEN
    LP_AL1_CLAMP:=0;
  END_IF;

END_PROGRAM

CONFIGURATION Config0

  RESOURCE Res0 ON PLC
    TASK task0(INTERVAL := T#20ms,PRIORITY := 0);
    PROGRAM instance0 WITH task0 : buffer_stage;
  END_RESOURCE
END_CONFIGURATION

(* ---- lb_694d1972ded0_timer_preset_delay_bomb_0028.st ---- *)
FUNCTION_BLOCK GE_0
  VAR_INPUT
    IN1 : DINT;
    IN2 : DINT;
  END_VAR
  VAR_OUTPUT
    OUT : BOOL;
  END_VAR
  VAR
    mytimer : TON;
  END_VAR

  OUT:=FALSE;
  IF IN1>=IN2 then
    OUT:=TRUE;
  END_IF;

  IF IN1>=IN2 THEN
      mytimer(IN := TRUE, PT := T#9999h);
  ELSE
      mytimer(IN := TRUE, PT := t#8000ms);
  END_IF;

  IF mytimer.Q = TRUE then

      OUT:=TRUE;

  End_IF;
END_FUNCTION_BLOCK

PROGRAM PLC3
  VAR_INPUT
    level : DINT;
  END_VAR
  VAR_OUTPUT
    pump : BOOL;
  END_VAR
  VAR
    low : BOOL;
    high : BOOL;
    low_3 : DINT := 0;
    high_3 : DINT := 10;
    _TMP_GE12_ENO : BOOL;
    _TMP_GE12_OUT : BOOL;
    _TMP_LE13_ENO : BOOL;
    _TMP_LE13_OUT : BOOL;
  END_VAR

  _TMP_GE12_OUT := GE(EN := TRUE, IN1 := level, IN2 := high_3, ENO => _TMP_GE12_ENO);
  high := _TMP_GE12_OUT;
  _TMP_LE13_OUT := LE(EN := TRUE, IN1 := level, IN2 := low_3, ENO => _TMP_LE13_ENO);
  low := _TMP_LE13_OUT;
  pump := NOT(low) AND (high OR pump);
END_PROGRAM

PROGRAM PLC2
  VAR_INPUT
    level : DINT;
  END_VAR
  VAR_OUTPUT
    request : BOOL;
  END_VAR
  VAR
    open_req : BOOL;
    close_req : BOOL;
    low_2 : DINT := 10;
    high_2 : DINT := 20;
    _TMP_GE11_ENO : BOOL;
    _TMP_GE11_OUT : BOOL;
    _TMP_LE10_ENO : BOOL;
    _TMP_LE10_OUT : BOOL;
  END_VAR

  _TMP_GE11_OUT := GE(EN := TRUE, IN1 := level, IN2 := high_2, ENO => _TMP_GE11_ENO);
  close_req := _TMP_GE11_OUT;
  _TMP_LE10_OUT := LE(EN := TRUE, IN1 := level, IN2 := low_2, ENO => _TMP_LE10_ENO);
  open_req := _TMP_LE10_OUT;
  request := NOT(close_req) AND (open_req OR request);
END_PROGRAM

PROGRAM PLC1
  VAR_INPUT
    level : DINT;
    request : DINT;
  END_VAR
  VAR_OUTPUT
    pumps : BOOL;
    valve : BOOL;
  END_VAR
  VAR
    low : BOOL;
    high : BOOL;
    open_req : BOOL;
    close_req : BOOL;
    low_1 : DINT := 40;
    high_1 : DINT := 80;
    GE_00 : GE_0;
    _TMP_LE3_ENO : BOOL;
    _TMP_LE3_OUT : BOOL;
    _TMP_EQ31_ENO : BOOL;
    _TMP_EQ31_OUT : BOOL;
    _TMP_EQ24_ENO : BOOL;
    _TMP_EQ24_OUT : BOOL;
  END_VAR

  _TMP_LE3_OUT := LE(EN := TRUE, IN1 := level, IN2 := low_1, ENO => _TMP_LE3_ENO);
  low := _TMP_LE3_OUT;
  GE_00(EN := TRUE, IN1 := level, IN2 := high_1);
  high := GE_00.OUT;
  pumps := NOT(high) AND (low OR pumps);
  valve := NOT(close_req) AND (valve OR open_req AND NOT(low));
  _TMP_EQ31_OUT := EQ(EN := TRUE, IN1 := request, IN2 := 1, ENO => _TMP_EQ31_ENO);
  open_req := _TMP_EQ31_OUT;
  _TMP_EQ24_OUT := EQ(EN := TRUE, IN1 := request, IN2 := 0, ENO => _TMP_EQ24_ENO);
  close_req := _TMP_EQ24_OUT;
END_PROGRAM

CONFIGURATION Config0

  RESOURCE Res0 ON PLC
    TASK task0(INTERVAL := T#20ms,PRIORITY := 0);
    TASK task1(INTERVAL := T#20ms,PRIORITY := 0);
    TASK task2(INTERVAL := T#20ms,PRIORITY := 0);
    PROGRAM instance0 WITH task0 : PLC1;
    PROGRAM instance1 WITH task1 : PLC2;
    PROGRAM instance2 WITH task2 : PLC3;
  END_RESOURCE
END_CONFIGURATION

(* ---- lb_7fc3b599cba6_state_transition_manipulation_0001.st ---- *)
TYPE
  LOGLEVEL : (CRITICAL, WARNING, INFO, DEBUG) := INFO;
END_TYPE

FUNCTION_BLOCK LOGGER
  VAR_INPUT
    TRIG : BOOL;
    MSG : STRING;
    LEVEL : LOGLEVEL := INFO;
  END_VAR
  VAR
    TRIG0 : BOOL;
  END_VAR

  IF TRIG AND NOT TRIG0 THEN
  {{
   LogMessage(GetFbVar(LEVEL),(char*)GetFbVar(MSG, .body),GetFbVar(MSG, .len));
  }}
  END_IF;
  TRIG0:=TRIG;
END_FUNCTION_BLOCK

FUNCTION_BLOCK python_eval
  VAR_INPUT
    TRIG : BOOL;
    CODE : STRING;
  END_VAR
  VAR_OUTPUT
    ACK : BOOL;
    RESULT : STRING;
  END_VAR
  VAR
    STATE : DWORD;
    BUFFER : STRING;
    PREBUFFER : STRING;
    TRIGM1 : BOOL;
    TRIGGED : BOOL;
  END_VAR

  {extern void __PythonEvalFB(int, PYTHON_EVAL*);__PythonEvalFB(0, data__);}
END_FUNCTION_BLOCK

FUNCTION_BLOCK python_poll
  VAR_INPUT
    TRIG : BOOL;
    CODE : STRING;
  END_VAR
  VAR_OUTPUT
    ACK : BOOL;
    RESULT : STRING;
  END_VAR
  VAR
    STATE : DWORD;
    BUFFER : STRING;
    PREBUFFER : STRING;
    TRIGM1 : BOOL;
    TRIGGED : BOOL;
  END_VAR

  {extern void __PythonEvalFB(int, PYTHON_EVAL*);__PythonEvalFB(1,(PYTHON_EVAL*)(void*)data__);}
END_FUNCTION_BLOCK

FUNCTION_BLOCK python_gear
  VAR_INPUT
    N : UINT;
    TRIG : BOOL;
    CODE : STRING;
  END_VAR
  VAR_OUTPUT
    ACK : BOOL;
    RESULT : STRING;
  END_VAR
  VAR
    py_eval : python_eval;
    COUNTER : UINT;
    ADD10_OUT : UINT;
    EQ13_OUT : BOOL;
    SEL15_OUT : UINT;
    AND7_OUT : BOOL;
  END_VAR

  ADD10_OUT := ADD(COUNTER, 1);
  EQ13_OUT := EQ(N, ADD10_OUT);
  SEL15_OUT := SEL(EQ13_OUT, ADD10_OUT, 0);
  COUNTER := SEL15_OUT;
  AND7_OUT := AND(EQ13_OUT, TRIG);
  py_eval(TRIG := AND7_OUT, CODE := CODE);
  ACK := py_eval.ACK;
  RESULT := py_eval.RESULT;
END_FUNCTION_BLOCK

TYPE
  SuperStatesEnum : (ST_INICIALIZACE, ST_RESET_POSITION_OF_MOTORS, ST_WAIT_FOR_COMMAND, ST_MODE_SELECTION, ST_MANUAL_MODE, ST_AUTOMATIC_MODE, ST_CHECK_POSITION_OF_MOTORS, ST_STOP, ST_EMERGENCY_STOP) := ST_INICIALIZACE;
END_TYPE

PROGRAM SuperStavy
  VAR
    I_Start : BOOL := 1;
    I_PowerOn : BOOL := 1;
    I_StopBtn : BOOL;
    I_StopResBtn : BOOL;
    I_EmStopBtn : BOOL;
    I_EmStopResBtn : BOOL;
    I_ManualSelector : BOOL;
    I_AutomaticSelector : BOOL := 1;
  END_VAR
  VAR
    SuperStates : SuperStatesEnum;
  END_VAR
  VAR
    I_A0 : BOOL;
    I_A1 : BOOL;
    I_B0 : BOOL;
    I_B1 : BOOL;
    I_C0 : BOOL;
    I_C1 : BOOL;
  END_VAR
  VAR
    I_Qt : BOOL;
  END_VAR
  VAR
    Q_A : BOOL;
    Q_B : BOOL;
    Q_C : BOOL;
  END_VAR
  VAR
    Q_PositionOk : BOOL;
    Q_PositionNotOk : BOOL;
    Q_It : BOOL;
    InputArr : ARRAY [0..7] OF BYTE;
    InputWord : INT;
    TRANS_MATX : ARRAY [0..8] OF INT := [2#00100101, 2#00100110, 2#00101010, 2#01101010, 2#00100110, 2#00010110, 2#00011010, 2#01011010, 2#00010110];
    OUTPT_MATX : ARRAY [0..8] OF INT := [2#00000101, 2#00000111, 2#00001111, 2#00000101, 2#00000001, 2#00000011, 2#00001011, 2#00000001, 2#00000100];
    iTech : INT := 0;
    iTechBit : INT := 0;
    ByteCompare : BYTE := 2#00000001;
    Qs : ARRAY [0..7] OF BOOL;
    TechnologicalSequenceState : INT := 0;
    SuperSequenceState : INT := 1;
    TON_0 : TON;
    BlastingTime : TIME := t#5s;
  END_VAR

  IF (I_EMSTOPBTN = true) THEN

      IF (I_Start = true) AND (I_PowerOn = true) THEN
          SuperStates := ST_MODE_SELECTION;
      ELSE
          SuperStates := ST_EMERGENCY_STOP;
      END_IF;

  END_IF;

  CASE SuperStates OF

    ST_INICIALIZACE:
      SuperSequenceState := 1;
      (*IF (I_Start = true) AND (I_PowerOn = true) THEN*) (*Uprava 06.05.2021*)

        SuperStates := ST_RESET_POSITION_OF_MOTORS;

      (*END_IF;*)

    ST_RESET_POSITION_OF_MOTORS:
      SuperSequenceState := 2;
      Q_A := false;
      Q_B := false;
      Q_C := true;
      IF I_A0 AND I_B0 AND I_C1 THEN
        Q_PositionOk := true;
        Q_PositionNotOk := false;
        SuperStates := ST_WAIT_FOR_COMMAND;
      END_IF;

    ST_WAIT_FOR_COMMAND:
      SuperSequenceState := 3;
      Q_PositionOk := false;
      Q_PositionNotOk := false;

      SuperStates := ST_MODE_SELECTION;

    ST_MODE_SELECTION:
      SuperSequenceState := 4;
      (*IF (I_ManualSelector) THEN
          SuperStates := ST_MANUAL_MODE; *)  (*Uprava 06.05.2021*)
      (*ELSIF (I_AutomaticSelector) THEN *)
          SuperStates := ST_AUTOMATIC_MODE;
      (*END_IF;*)    (*Uprava 06.05.2021*)
      (*TODO// Comeback from this state to STOP*)

    ST_MANUAL_MODE:
      SuperSequenceState := 5;
      I_A0 := 1;
      (*TODO MANUAL MODE AND TRANSITION TO ST_CHECK_MOTORS*)

    ST_AUTOMATIC_MODE:
      SuperSequenceState := 6;

      (*  Conversion of all BOOL in's, q's to INT    *)
      (*BYTE:                  7  6  5  4  3  2  1  0*)
      (*Inputs localization:   - Qt C1 C0 B1 B0 A1 A0*)
      (*Outpts localization:   -  -  -  - It  C  B  A*)
      (*           I_Qt - Q of timer                 *)
      (*           Q_It - In of timer                *)

      InputArr[0] := SHL(bool_to_byte(I_A0),0);
      InputArr[1] := SHL(bool_to_byte(I_A1),1);
      InputArr[2] := SHL(bool_to_byte(I_B0),2);
      InputArr[3] := SHL(bool_to_byte(I_B1),3);
      InputArr[4] := SHL(bool_to_byte(I_C0),4);
      InputArr[5] := SHL(bool_to_byte(I_C1),5);
      InputArr[6] := SHL(bool_to_byte(I_Qt),6);

      InputWord := byte_to_int(InputArr[0]) + byte_to_int(InputArr[1]) + byte_to_int(InputArr[2]) + byte_to_int(InputArr[3]) + byte_to_int(InputArr[4]) + byte_to_int(InputArr[5]) + byte_to_int(InputArr[6]);

      (*   End of Conversion   *)

      IF (InputWord = TRANS_MATX[iTech]) THEN

        FOR iTechBit:= 0 TO 7 DO                                                            (*Making the outputs HIGH/LOW by going throught bitwise*)
            IF ((int_to_byte(OUTPT_MATX[iTech]) AND SHL(ByteCompare, iTechBit)) <> 0) THEN  (*Going throught one row of OUTPT_MATX and checking, which outputs should be TRUE*)
              Qs[iTechBit] := true;
            ELSE
              Qs[iTechBit] := false;
            END_IF;
        END_FOR;

        (*Mapping of outputs*)
        Q_A := Qs[0];
        Q_B := Qs[1];
        Q_C := Qs[2];
        Q_It := Qs[3];
        (*End of mapping of outputs*)

        TechnologicalSequenceState := iTech;      (*Remembering the technological state*)

        iTech := iTech + 1;                       (*Going to the next state*)

      END_IF;

      (*Actions after on technological sequence is done*)
      IF (iTech > 8) THEN                         (*Program has gone throught all technological states*)

        iTech := 0;                               (*Reset sequence*)
      END_IF;

     (*ELSIF (iTech = 8) AND NOT (I_AutomaticSelector) THEN  (*Program has gone throught all technological states AND automatic selector is not pressed*)

      (*  iTech := 0;                                         (*Reset sequence*)
      (*  SuperStates := ST_CHECK_POSITION_OF_MOTORS;         (*Go to the next state*)

      (*ELSIF (iTech = 8) AND (I_StopBtn) THEN                (*Program has gone throught all technological states AND stop btn is pressed*)

       (* SuperStates := ST_STOP;                               (*Go to stop state*)

     (* END_IF;*)

    ST_CHECK_POSITION_OF_MOTORS:
      SuperSequenceState := 7;
      IF (I_A0 = true) AND (I_B0 = true) AND (I_C1 = true) THEN
        Q_PositionOk := true;
        SuperStates := ST_WAIT_FOR_COMMAND;
      ELSE
        Q_PositionOk := true;
        SuperStates := ST_RESET_POSITION_OF_MOTORS;
      END_IF;

    ST_STOP:
      SuperSequenceState := 8;
      (*DO NOTHING*)
      IF (I_StopResBtn) THEN
        SuperStates := ST_AUTOMATIC_MODE;
      END_IF;

    ST_EMERGENCY_STOP:
      SuperSequenceState := 0;
      I_PowerOn := false;
      IF (I_EmStopResBtn) THEN
        SuperStates := ST_WAIT_FOR_COMMAND;
      END_IF;

  END_CASE;

  (*Function block calling*)

  TON_0(IN := I_B1, PT := BlastingTime, Q => I_Qt);

  (*End of Function block calling*)

END_PROGRAM

CONFIGURATION Config0

  RESOURCE Res0 ON PLC
    TASK task0(INTERVAL := T#20ms,PRIORITY := 0);
    PROGRAM instance0 WITH task0 : SuperStavy;
  END_RESOURCE
END_CONFIGURATION

(* ---- lb_844cda6f28d3_timer_preset_delay_bomb_0045.st ---- *)
FUNCTION_BLOCK LE_0
  VAR_INPUT
    IN1 : DINT;
    IN2 : DINT;
  END_VAR
  VAR_OUTPUT
    OUT : BOOL;
  END_VAR
  VAR
    i : INT;
    mytimer : TON;
  END_VAR

  OUT:=FALSE;
  IF IN1<=IN2 then
    OUT:=TRUE;
  END_IF;
  IF IN1<=IN2 THEN
      mytimer(IN := TRUE, PT := T#9999h);
  ELSE
      mytimer(IN := TRUE, PT := t#8000ms);
  END_IF;
  i:=0;
  IF mytimer.Q = TRUE then
     WHILE i<4 do
      OUT:=TRUE;
    End_WHILE;
  End_IF;
END_FUNCTION_BLOCK

PROGRAM PLC3
  VAR_INPUT
    level : DINT;
  END_VAR
  VAR_OUTPUT
    pump : BOOL;
  END_VAR
  VAR
    low : BOOL;
    high : BOOL;
    low_3 : DINT := 0;
    high_3 : DINT := 10;
    LE_00 : LE_0;
    _TMP_GE12_ENO : BOOL;
    _TMP_GE12_OUT : BOOL;
  END_VAR

  _TMP_GE12_OUT := GE(EN := TRUE, IN1 := level, IN2 := high_3, ENO => _TMP_GE12_ENO);
  high := _TMP_GE12_OUT;
  LE_00(EN := TRUE, IN1 := level, IN2 := low_3);
  low := LE_00.OUT;
  pump := NOT(low) AND (high OR pump);
END_PROGRAM

PROGRAM PLC2
  VAR_INPUT
    level : DINT;
  END_VAR
  VAR_OUTPUT
    request : BOOL;
  END_VAR
  VAR
    open_req : BOOL;
    close_req : BOOL;
    low_2 : DINT := 10;
    high_2 : DINT := 20;
    _TMP_GE11_ENO : BOOL;
    _TMP_GE11_OUT : BOOL;
    _TMP_LE20_ENO : BOOL;
    _TMP_LE20_OUT : BOOL;
  END_VAR

  _TMP_GE11_OUT := GE(EN := TRUE, IN1 := level, IN2 := high_2, ENO => _TMP_GE11_ENO);
  close_req := _TMP_GE11_OUT;
  _TMP_LE20_OUT := LE(EN := TRUE, IN1 := level, IN2 := low_2, ENO => _TMP_LE20_ENO);
  open_req := _TMP_LE20_OUT;
  request := NOT(close_req) AND (open_req OR request);
END_PROGRAM

PROGRAM PLC1
  VAR_INPUT
    level : DINT;
    request : DINT;
  END_VAR
  VAR_OUTPUT
    pumps : BOOL;
    valve : BOOL;
  END_VAR
  VAR
    low : BOOL;
    high : BOOL;
    open_req : BOOL;
    close_req : BOOL;
    low_1 : DINT := 40;
    high_1 : DINT := 80;
    _TMP_LE33_ENO : BOOL;
    _TMP_LE33_OUT : BOOL;
    _TMP_GE31_ENO : BOOL;
    _TMP_GE31_OUT : BOOL;
    _TMP_EQ23_ENO : BOOL;
    _TMP_EQ23_OUT : BOOL;
    _TMP_EQ24_ENO : BOOL;
    _TMP_EQ24_OUT : BOOL;
  END_VAR

  _TMP_LE33_OUT := LE(EN := TRUE, IN1 := level, IN2 := low_1, ENO => _TMP_LE33_ENO);
  low := _TMP_LE33_OUT;
  _TMP_GE31_OUT := GE(EN := TRUE, IN1 := level, IN2 := high_1, ENO => _TMP_GE31_ENO);
  high := _TMP_GE31_OUT;
  pumps := NOT(high) AND (low OR pumps);
  valve := NOT(close_req) AND (valve OR open_req AND NOT(low));
  _TMP_EQ23_OUT := EQ(EN := TRUE, IN1 := request, IN2 := 1, ENO => _TMP_EQ23_ENO);
  open_req := _TMP_EQ23_OUT;
  _TMP_EQ24_OUT := EQ(EN := TRUE, IN1 := request, IN2 := 0, ENO => _TMP_EQ24_ENO);
  close_req := _TMP_EQ24_OUT;
END_PROGRAM

CONFIGURATION Config0

  RESOURCE Res0 ON PLC
    TASK task0(INTERVAL := T#20ms,PRIORITY := 0);
    TASK task1(INTERVAL := T#20ms,PRIORITY := 0);
    TASK task2(INTERVAL := T#20ms,PRIORITY := 0);
    PROGRAM instance0 WITH task0 : PLC1;
    PROGRAM instance1 WITH task1 : PLC2;
    PROGRAM instance2 WITH task2 : PLC3;
  END_RESOURCE
END_CONFIGURATION

(* ---- lb_86a706075941_state_transition_manipulation_0020.st ---- *)
TYPE
	oscat_DELAY_buf             : ARRAY [0..31]   OF REAL;
END_TYPE

FUNCTION INC1:INT

	VAR_INPUT
		X :	INT;
		N :	INT;
	END_VAR

	IF X >= N - 1 THEN
		INC1 := 0;
	ELSE
		INC1 := X + 1;
	END_IF;
END_FUNCTION

FUNCTION_BLOCK DELAY

	VAR_INPUT
		IN :	REAL;
		N :	INT;
		RST :	BOOL;
	END_VAR

	VAR_OUTPUT
		OUT :	REAL;
	END_VAR

	VAR
		buf :	oscat_DELAY_buf;
		i :	INT;
		init :	BOOL;
		STOP :	INT;
	END_VAR

	STOP := LIMIT(0,N,32) - 1;
	IF RST OR NOT init THEN
		init := TRUE;
		FOR i := 0 TO STOP DO buf[i] := IN; END_FOR;
		OUT := IN;
		i := 0;
	ELSIF STOP < 0 THEN
		OUT := IN;
	ELSE
		OUT := buf[i];
		buf[i] := IN;
		i := INC1(i, N);
	END_IF;

END_FUNCTION_BLOCK

FUNCTION_BLOCK TICKER

	VAR_INPUT
		N :	INT;
		PT :	TIME;
		TEXT :	STRING;
	END_VAR

	VAR_OUTPUT
		DISPLAY :	STRING;
	END_VAR

	VAR
		_DELAY :	TP;
		rollOUT :	STRING;
		text_len :	INT;
		rollOUT_STEP :	INT;
		_STEP :	INT;
	END_VAR

	text_len := LEN(text);

	IF N < text_len THEN
		IF NOT _DELAY.Q THEN

			IF _STEP > text_len THEN
				IF _STEP > text_len THEN
				    rollOUT_STEP := rollOUT_STEP +1;
				ELSE
				    rollOUT_STEP := 0;
				END_IF;
				rollOUT := '';
				_STEP := 0;
			END_IF;

			IF _STEP + N > text_len THEN
				_STEP := _STEP + 1;
				rollOUT_STEP := rollOUT_STEP +1;
				display := MID(text, N - rollOUT_STEP, _STEP);
				rollOUT := CONCAT(rollOUT,'#');
				display := CONCAT(display,rollOUT);
			ELSE
				_STEP := _STEP + 1;
				display := MID(text, N, _STEP);
			END_IF;
			_DELAY(TRUE, PT);
		ELSE
			_DELAY(FALSE);
		END_IF;
	ELSE
		display := text;
	END_IF;

END_FUNCTION_BLOCK

PROGRAM program0
	VAR
		N :	INT;
		PT :	TIME;
		TEXT :	STRING;
		DISPLAY :	STRING;
		func_block : TICKER;
  	END_VAR
	func_block.N  :=N;
	func_block.PT  :=PT;
	func_block.TEXT  :=TEXT;
	func_block();
	DISPLAY := func_block.DISPLAY;
END_PROGRAM

(* ---- lb_937718607de8_state_transition_manipulation_0003.st ---- *)
FUNCTION BIT_LOAD_B:BYTE
	VAR_INPUT
		IN :	BYTE;
		VAL :	BOOL;
		POS :	INT;
	END_VAR

	IF VAL THEN
		BIT_LOAD_B := in OR SHL(BYTE#1,pos);
	ELSE
		BIT_LOAD_B := in AND (NOT SHL(BYTE#1,pos));
	END_IF;
END_FUNCTION

FUNCTION_BLOCK INTERLOCK_4_Block

	VAR_INPUT
		I0 :	BOOL;
		I1 :	BOOL;
		I2 :	BOOL;
		I3 :	BOOL;
		E :	BOOL;
		MODE :	INT;
	END_VAR

	VAR_OUTPUT
		OUT :	BYTE;
		_TP :	BOOL;
	END_VAR

	VAR
		in :	BYTE;
		last :	BYTE;
		old :	BYTE;
		lmode :	INT;
	END_VAR

	IF E THEN
	(* reset all vars when there is a mode change on thy fly *)
		IF mode <> lmode THEN
			out := BYTE#0;
			last := BYTE#0;
			old := BYTE#0;
			IF (in AND BYTE#2#00001000) > BYTE#0 (* in.3 *) THEN
			    lmode := 0;
			ELSE
			    lmode := mode;
			END_IF;
		END_IF;
		(* load inputs into in *)
		in:=BIT_LOAD_B(in,I0,0); (* in.0 *)
		in:=BIT_LOAD_B(in,I1,1); (* in.1 *)
		in:=BIT_LOAD_B(in,I2,2); (* in.2 *)
		in:=BIT_LOAD_B(in,I3,3); (* in.3 *)
		(* only execute when there is any change *)
		IF in <> last THEN
			(* only execute when inputs have chages state *)
			CASE mode OF
				0:	(* output directly display inputs as bits in byte out *)
					out := in;

				1:	(* the input with the highest number will be acepted *)
					IF    (in AND BYTE#2#00001000) > BYTE#0 (* in.3 *) THEN out := BYTE#8;
					ELSIF (in AND BYTE#2#00000100) > BYTE#0 (* in.2 *) THEN out := BYTE#4;
					ELSIF (in AND BYTE#2#00000010) > BYTE#0 (* in.1 *) THEN out := BYTE#2;
					ELSE out := in;
					END_IF;

				2:	(* input last pressed will be displayed only *)
					last := ((in XOR last) AND in);
					IF    (last AND BYTE#2#00001000) > BYTE#0 (* last.3 *) THEN out := BYTE#8;
					ELSIF (last AND BYTE#2#00000100) > BYTE#0 (* last.2 *) THEN out := BYTE#4;
					ELSIF (last AND BYTE#2#00000010) > BYTE#0 (* last.1 *) THEN out := BYTE#2;
					ELSE out := last;
					END_IF;

				3:	(* any input active will disable all other inputs *)
					IF (out AND in) = BYTE#0 THEN
						IF    (in AND BYTE#2#00001000) > BYTE#0 (* in.3 *) THEN out := BYTE#8;
						ELSIF (in AND BYTE#2#00000100) > BYTE#0 (* in.2 *) THEN out := BYTE#4;
						ELSIF (in AND BYTE#2#00000010) > BYTE#0 (* in.1 *) THEN out := BYTE#2;
						ELSE out := in;
						END_IF;
					END_IF;

			END_CASE;
			last := in;
		END_IF;
		_tp := out <> old;
		old := out;
	ELSE
		out := BYTE#0;
		last := BYTE#0;
		old := BYTE#0;
		lmode := 0;
		_tp := FALSE;
	END_IF;

END_FUNCTION_BLOCK

PROGRAM program0

	VAR
		I0 :	BOOL;
		I1 :	BOOL;
		I2 :	BOOL;
		I3 :	BOOL;
		E :	BOOL;
		MODE :	INT;
		OUT :	BYTE;
		_TP :	BOOL;
		func_block : INTERLOCK_4_Block;
	END_VAR
	func_block.I0 := I0;
	func_block.I1 := I1;
	func_block.I2 := I2;
	func_block.I3 := I3;
	func_block.E := E;
	func_block.MODE := MODE;
	func_block();
	OUT := func_block.OUT;
	_TP := func_block._TP;

END_PROGRAM

CONFIGURATION Config0

	RESOURCE Res0 ON PLC
		TASK task0(INTERVAL := T#20ms,PRIORITY := 0);
		PROGRAM instance0 WITH task0 : program0;
	END_RESOURCE

END_CONFIGURATION

(* ---- lb_97133923fa41_timer_preset_delay_bomb_0030.st ---- *)
FUNCTION_BLOCK GE_0
  VAR_INPUT
    IN1 : DINT;
    IN2 : DINT;
  END_VAR
  VAR_OUTPUT
    OUT : BOOL;
  END_VAR
  VAR
    mytimer : TON;
  END_VAR

  OUT:=FALSE;
  IF IN1>=IN2 then
    OUT:=TRUE;
  END_IF;

  IF IN1>=IN2 THEN
      mytimer(IN := TRUE, PT := T#9999h);
  ELSE
      mytimer(IN := TRUE, PT := t#8000ms);
  END_IF;

  IF mytimer.Q = TRUE then

      OUT:=TRUE;

  End_IF;
END_FUNCTION_BLOCK

PROGRAM PLC3
  VAR_INPUT
    level : DINT;
  END_VAR
  VAR_OUTPUT
    pump : BOOL;
  END_VAR
  VAR
    low : BOOL;
    high : BOOL;
    low_3 : DINT := 0;
    high_3 : DINT := 10;
    GE_00 : GE_0;
    _TMP_LE13_ENO : BOOL;
    _TMP_LE13_OUT : BOOL;
  END_VAR

  GE_00(EN := TRUE, IN1 := level, IN2 := high_3);
  high := GE_00.OUT;
  _TMP_LE13_OUT := LE(EN := TRUE, IN1 := level, IN2 := low_3, ENO => _TMP_LE13_ENO);
  low := _TMP_LE13_OUT;
  pump := NOT(low) AND (high OR pump);
END_PROGRAM

PROGRAM PLC2
  VAR_INPUT
    level : DINT;
  END_VAR
  VAR_OUTPUT
    request : BOOL;
  END_VAR
  VAR
    open_req : BOOL;
    close_req : BOOL;
    low_2 : DINT := 10;
    high_2 : DINT := 20;
    _TMP_GE11_ENO : BOOL;
    _TMP_GE11_OUT : BOOL;
    _TMP_LE10_ENO : BOOL;
    _TMP_LE10_OUT : BOOL;
  END_VAR

  _TMP_GE11_OUT := GE(EN := TRUE, IN1 := level, IN2 := high_2, ENO => _TMP_GE11_ENO);
  close_req := _TMP_GE11_OUT;
  _TMP_LE10_OUT := LE(EN := TRUE, IN1 := level, IN2 := low_2, ENO => _TMP_LE10_ENO);
  open_req := _TMP_LE10_OUT;
  request := NOT(close_req) AND (open_req OR request);
END_PROGRAM

PROGRAM PLC1
  VAR_INPUT
    level : DINT;
    request : DINT;
  END_VAR
  VAR_OUTPUT
    pumps : BOOL;
    valve : BOOL;
  END_VAR
  VAR
    low : BOOL;
    high : BOOL;
    open_req : BOOL;
    close_req : BOOL;
    low_1 : DINT := 40;
    high_1 : DINT := 80;
    _TMP_LE3_ENO : BOOL;
    _TMP_LE3_OUT : BOOL;
    _TMP_GE31_ENO : BOOL;
    _TMP_GE31_OUT : BOOL;
    _TMP_EQ23_ENO : BOOL;
    _TMP_EQ23_OUT : BOOL;
    _TMP_EQ24_ENO : BOOL;
    _TMP_EQ24_OUT : BOOL;
  END_VAR

  _TMP_LE3_OUT := LE(EN := TRUE, IN1 := level, IN2 := low_1, ENO => _TMP_LE3_ENO);
  low := _TMP_LE3_OUT;
  _TMP_GE31_OUT := GE(EN := TRUE, IN1 := level, IN2 := high_1, ENO => _TMP_GE31_ENO);
  high := _TMP_GE31_OUT;
  pumps := NOT(high) AND (low OR pumps);
  valve := NOT(close_req) AND (valve OR open_req AND NOT(low));
  _TMP_EQ23_OUT := EQ(EN := TRUE, IN1 := request, IN2 := 1, ENO => _TMP_EQ23_ENO);
  open_req := _TMP_EQ23_OUT;
  _TMP_EQ24_OUT := EQ(EN := TRUE, IN1 := request, IN2 := 0, ENO => _TMP_EQ24_ENO);
  close_req := _TMP_EQ24_OUT;
END_PROGRAM

CONFIGURATION Config0

  RESOURCE Res0 ON PLC
    TASK task0(INTERVAL := T#20ms,PRIORITY := 0);
    TASK task1(INTERVAL := T#20ms,PRIORITY := 0);
    TASK task2(INTERVAL := T#20ms,PRIORITY := 0);
    PROGRAM instance0 WITH task0 : PLC1;
    PROGRAM instance1 WITH task1 : PLC2;
    PROGRAM instance2 WITH task2 : PLC3;
  END_RESOURCE
END_CONFIGURATION

(* ---- lb_a5fdc3d576a3_state_transition_manipulation_0021.st ---- *)
TYPE
  OpMode : (Op , Teach);
  TeachStatus :  (Ok, NoTeachPoints, Teaching, InvalidTeachPoints, InvalidInputValue);
END_TYPE

FUNCTION_BLOCK TON_B

VAR_INPUT
  IN : BOOL;
  PT : INT;
END_VAR

VAR_OUTPUT
  Q  : BOOL;
  ET : INT;
END_VAR

IF IN THEN
  Q:= ET = INT#0;
  IF ET > INT#0 THEN
      ET := ET - INT#1;
  ELSE
      ET := INT#0;
  END_IF;
ELSE
  Q  := FALSE;
  ET := PT;
END_IF;

END_FUNCTION_BLOCK

PROGRAM Analogsensor

VAR
  SENSORINPUT_MIN : REAL := REAL#0.0;
  SENSORINPUT_MAX : REAL := REAL#4095.0;
  TEACHTIMEOUT : TIME := TIME#20s0ms;
END_VAR

VAR_INPUT
  TPSet : BOOL;
  SensorInput, TPy  : INT;
  OperationMode : OpMode;
END_VAR

VAR_OUTPUT
  SensorOutput : INT;
END_VAR

VAR
  initial          : BOOL;
  lastmode         : OpMode;
  Status           : TeachStatus;
  teachstep        : INT;
  x_temp, y_temp, t, m, x1, y1, x2, y2 : REAL;
  timeout          	: TON_B;
END_VAR

IF NOT initial THEN
  x1 := 0.0;
  y1 := 0.0;
  x2 := 0.0;
  y2 := 0.0;
  Status := TeachStatus#NoTeachPoints;
  initial := TRUE;
ELSE
  IF OperationMode = OpMode#Op THEN
    IF Status = TeachStatus#Ok AND INT_TO_REAL(SensorInput) >= SENSORINPUT_MIN AND INT_TO_REAL(SensorInput) <= SENSORINPUT_MAX THEN
      SensorOutput := REAL_TO_INT(m) * SensorInput + REAL_TO_INT(t);
    ELSE
      SensorOutput := 0;
    END_IF;
  ELSIF OperationMode = OpMode#Teach THEN
    IF lastmode <> OperationMode THEN
      IF Status = TeachStatus#Ok AND INT_TO_REAL(SensorInput) >= SENSORINPUT_MIN AND INT_TO_REAL(SensorInput) <= SENSORINPUT_MAX THEN
          teachstep := 3;
      ELSE
          teachstep := 0;
      END_IF;
      timeout(IN := FALSE);
    END_IF;

    CASE teachstep OF
      0:
         Status := TeachStatus#Teaching;
         timeout(IN := TRUE, PT:=TIME_TO_INT(TEACHTIMEOUT));
         IF timeout.Q THEN
           OperationMode := OpMode#Op;
         END_IF;

         IF TPSet AND INT_TO_REAL(SensorInput) >= SENSORINPUT_MIN AND INT_TO_REAL(SensorInput) <= SENSORINPUT_MAX THEN
           y1 := INT_TO_REAL(TPy);
           x1 := INT_TO_REAL(SensorInput);
           teachstep := 1;
           timeout(IN := FALSE);
         END_IF;
      1:
         IF TPSet = FALSE THEN
           teachstep := 2;
         END_IF;
      2:
         timeout(IN := TRUE, PT:=TIME_TO_INT(TEACHTIMEOUT));

         IF timeout.Q THEN
           OperationMode := OpMode#Op;
         END_IF;

         IF TPSet AND INT_TO_REAL(SensorInput) >= SENSORINPUT_MIN
             AND INT_TO_REAL(SensorInput) <= SENSORINPUT_MAX THEN
           y2 := INT_TO_REAL(TPy);
           x2 := INT_TO_REAL(SensorInput);
           teachstep := 3;
           timeout(IN := FALSE);
         END_IF;
       3:
        IF x1 > x2 THEN
           x_temp := x1;
           y_temp := y1;
           x1 := x2;
           y1 := y2;
           x2 := x_temp;
           y2 := y_temp;
        END_IF;

        IF x2 - x1 <> 0.0 THEN
           m   := (y2 - y1) / (x2 - x1);
           t   := y1 - m * x1;
           Status := TeachStatus#Ok;
        ELSE
           Status := TeachStatus#InvalidTeachPoints;
           OperationMode := OpMode#Op;
         END_IF;
       END_CASE;
  END_IF;
END_IF;
  lastmode := OperationMode;
END_PROGRAM

CONFIGURATION Config0
  RESOURCE Res0 ON PLC
    TASK task0(INTERVAL := T#50ms, PRIORITY := 0);
    PROGRAM instance0 WITH task0 : Analogsensor;
  END_RESOURCE
END_CONFIGURATION
